// TIA Portal project "Abschulss_Projekt" (V18)
// Vorlageprojekt für das Buch mit Zielsystem S7-1200

(* hardware
DEVICE "S7-1500/ET200MP-Station_1"  S7-1500 station
   slot 0: "Profilschiene_0"  Rack  6ES7 590-1***0-0AA0
   slot 1: "PLC_1"  CPU 1511-1 PN  6ES7 511-1AK00-0AB0  V1.8
      slot 3: "CPU-Display_1"  6ES7591-1AA00-0AA0
      slot 32768: "PROFINET-Schnittstelle_1"  X1
         slot 32769: "Port_1"  X1 P1
         slot 32770: "Port_2"  X1 P2
DEVICE "HMI_1"  KTP900 Basic PN
   slot 0: "HMI_1"  KTP900 Basic PN  6AV2 123-2JB03-0AX0  17.0.0.0
   slot 1: "HMI_RT_1"  KTP900 Basic PN  6AV2 123-2JB03-0AX0  17.0.0.0
   slot 5: "HMI_1.IE_CP_1"  PROFINET Interface  17.0.0.0
      slot 1: "PROFINET Schnittstelle_1"  PROFINET Interface
         slot 1: "Port_1"  Port
*)

// ===== PLC "PLC_1"  CPU 1511-1 PN =====

VAR_GLOBAL   // PLC tag table "Aktor"
   "FACTORY I/O (Reset)(1)" AT %Q8.0 : Bool;
   "Band_Base_1" AT %Q0.0 : Bool;
   "Band_Base_2" AT %Q0.1 : Bool;
   "Band_Base_4" AT %Q0.2 : Bool;
   "Band_Base_6_Gripper" AT %Q0.3 : Bool;
   "R1_Warning_Light" AT %Q0.4 : Bool;
   "R2_Warning_Light" AT %Q0.5 : Bool;
   "Band_Lid_1" AT %Q1.0 : Bool;
   "Band_Lid_2" AT %Q1.1 : Bool;
   "Band_Lid_4" AT %Q1.2 : Bool;
   "Band_Lid_6_Gripper" AT %Q1.3 : Bool;
   "Band_Palletizer_1" AT %Q1.4 : Bool;
   "Loading_to_Crane_Conveyor" AT %Q1.5 : Bool;
   "Emitter_Euro_Palette" AT %Q1.6 : Bool;
   "Curved_Band_Base_3" AT %Q1.7 : Bool;
   "Curved_Band_Base_5" AT %Q2.0 : Bool;
   "Curved_Band_Lid_3" AT %Q2.1 : Bool;
   "Curved_Band_Lid_5" AT %Q2.2 : Bool;
   "Emitter_Base" AT %Q2.3 : Bool;
   "Emitter_Lid" AT %Q2.4 : Bool;
   "Emitter_Package_M" AT %Q2.5 : Bool;
   "Grip_Gripper" AT %Q2.6 : Bool;
   "Palletizer_1_Push" AT %Q2.7 : Bool;
   "Palletizer_1_Turn" AT %Q3.0 : Bool;
   "Palletizer_1_Clamp" AT %Q3.1 : Bool;
   "Palletizer_1_Belt_Plus" AT %Q3.2 : Bool;
   "Palletizer_1_Chain_Plus" AT %Q3.3 : Bool;
   "Palletizer_1_Open_Plate" AT %Q3.4 : Bool;
   "Palletizer_1_Belt_Minuns" AT %Q3.5 : Bool;
   "Palletizer_1_Chain_Minus" AT %Q3.6 : Bool;
   "Palletizer_1_Elevator_Plus" AT %Q3.7 : Bool;
   "Palletizer_1_Elevator_Minus" AT %Q4.0 : Bool;
   "Palletizer_1_Elevator_Move_to_Limit" AT %Q4.1 : Bool;
   "Press_Base" AT %Q4.2 : Bool;
   "Press_Base_Positioner_0_Raise" AT %Q4.3 : Bool;
   "Press_Lid" AT %Q4.4 : Bool;
   "Press_Lid_Positioner_0_Raise" AT %Q4.5 : Bool;
   "R1_Stop" AT %Q4.6 : Bool;
   "R2_Stop" AT %Q4.7 : Bool;
   "R1_Reset" AT %Q5.0 : Bool;
   "R1_Start" AT %Q5.1 : Bool;
   "R2_Reset" AT %Q5.2 : Bool;
   "R2_Start" AT %Q5.3 : Bool;
   "R1_Produce_Lids" AT %Q5.4 : Bool;
   "R2_Produce_Base" AT %Q5.5 : Bool;
   "Remover_Product" AT %Q5.6 : Bool;
   "StackerCrane_1_Left" AT %Q5.7 : Bool;
   "StackerCrane_1_Lift" AT %Q6.0 : Bool;
   "StackerCrane_1_Right" AT %Q6.1 : Bool;
   "X_Move_Gripper" AT %Q6.2 : Bool;
   "Z_Move_Gripper" AT %Q6.3 : Bool;
   "StackerCrane_1_Target_1_Position" AT %QD100 : DInt;
   "Loading_Conveyor_Remover" AT %Q6.4 : Bool;
   "Remove_Euro_Palete" AT %Q6.5 : Bool;
END_VAR

VAR_GLOBAL   // PLC tag table "Merker"
   "Reset" AT %M15.0 : Bool;
END_VAR

VAR_GLOBAL   // PLC tag table "Sensor"
   "FACTORY I/O (Reset)" AT %I4.2 : Bool;
   "LT_Colour_Sorter" AT %I0.0 : Bool;
   "LT_Emitter_Base" AT %I0.1 : Bool;
   "LT_Emitter_Lid" AT %I0.2 : Bool;
   "LT_Palletizer" AT %I0.3 : Bool;
   "LT_Press_Base_Gripper" AT %I0.4 : Bool;
   "LT_Press_Lid_Gripper" AT %I0.5 : Bool;
   "Palletizer_1_Clamped" AT %I0.6 : Bool;
   "Palletizer_1_Plate_Limit" AT %I0.7 : Bool;
   "Palletizer_1_Pusher_Limit" AT %I1.0 : Bool;
   "Palletizer_1_Elevator_Moving" AT %I1.1 : Bool;
   "Palletizer_1_Elevator_Back_Limit" AT %I1.2 : Bool;
   "Palletizer_1_Elevator_Front_Limit" AT %I1.3 : Bool;
   "Press_Base_Positioner_0_Limit" AT %I1.4 : Bool;
   "Press_Lid_Positioner_0_Limit" AT %I1.5 : Bool;
   "R1_Opened" AT %I1.6 : Bool;
   "R2_Opened" AT %I1.7 : Bool;
   "R1_Is_Busy" AT %I2.0 : Bool;
   "R2_Is_Busy" AT %I2.1 : Bool;
   "R1_Has_Error" AT %I2.2 : Bool;
   "R2_Has_Error" AT %I2.3 : Bool;
   "Sensor_Base_fixiert" AT %I2.4 : Bool;
   "Sensor_Greifer_Teilerkennung" AT %I2.5 : Bool;
   "Sensor_Lid_fixiert" AT %I2.6 : Bool;
   "StackerCrane_1_Moving_X" AT %I2.7 : Bool;
   "StackerCrane_1_Moving_Z" AT %I3.0 : Bool;
   "StackerCrane_1_Left_Limit" AT %I3.1 : Bool;
   "StackerCrane_1_Right_Limit" AT %I3.2 : Bool;
   "X_Move_Sensor" AT %I3.3 : Bool;
   "Z_Move_Sensor" AT %I3.4 : Bool;
   "LT_Crane_Feed" AT %I3.5 : Bool;
   "StackerCrane_1_Middle_Limit" AT %I3.6 : Bool;
   "R1_Progress" AT %ID100 : DInt;
   "R2_Progress" AT %ID104 : DInt;
   "Vision_Sensor_Base" AT %ID108 : DInt;
   "Vision_Sensor_Lid" AT %ID112 : DInt;
   "LT_Remove_Palete" AT %I3.7 : Bool;
END_VAR

// folder: 01_Common

DATA_BLOCK "FB_Reset PLC und FactoryIO_DB"   // DB1
{ S7_Optimized_Access := 'TRUE' }
VERSION : 0.1
// stored: InstanceOfName FB_Reset PLC und FactoryIO
"FB_Reset PLC und FactoryIO"
BEGIN
END_DATA_BLOCK

DATA_BLOCK "DB_Global"   // DB2
{ S7_Optimized_Access := 'TRUE' }
VERSION : 0.1
   VAR
      Plant_Enabled : Bool := false;
      Warehouse_Full : Bool;
      Production_Enable : Bool;
      HMI_LidStatus : USInt;
      HMI_BaseStatus : USInt;
      HMI_WarehouseStatus : USInt;
      HMI_Status_OK : Bool;
      HMI_OccupiedPositions : DInt;
      HMI_FreePositions : DInt;
      HMI_TotalPackages : DInt;
      HMI_AlarmWord : Word;
      HMI_AckWord : Word;
   END_VAR
BEGIN
END_DATA_BLOCK

DATA_BLOCK "FB_ProductTracking_DB"   // DB3
{ S7_Optimized_Access := 'TRUE' }
VERSION : 0.1
// stored: InstanceOfName FB_ProductTracking
"FB_ProductTracking"
BEGIN
END_DATA_BLOCK

// folder: 02_Production

DATA_BLOCK "FB_LidCenter_DB"   // DB9
{ S7_Optimized_Access := 'TRUE' }
VERSION : 0.1
// stored: InstanceOfName FB_LidProduction
"FB_LidProduction"
BEGIN
END_DATA_BLOCK

DATA_BLOCK "FB_BaseCenter_DB"   // DB10
{ S7_Optimized_Access := 'TRUE' }
VERSION : 0.1
// stored: InstanceOfName FB_BaseProduction
"FB_BaseProduction"
BEGIN
END_DATA_BLOCK

// folder: 03_Assembly

DATA_BLOCK "FB_Assembly_DB"   // DB11
{ S7_Optimized_Access := 'TRUE' }
VERSION : 0.1
// stored: InstanceOfName FB_Assembly
"FB_Assembly"
BEGIN
END_DATA_BLOCK

DATA_BLOCK "FB_AssemblyActors_DB"   // DB12
{ S7_Optimized_Access := 'TRUE' }
VERSION : 0.1
// stored: InstanceOfName FB_AssemblyActors
"FB_AssemblyActors"
BEGIN
END_DATA_BLOCK

// folder: 04_Palletizer

DATA_BLOCK "FB_Palletizer_DB"   // DB13
{ S7_Optimized_Access := 'TRUE' }
VERSION : 0.1
// stored: InstanceOfName FB_Palletizer
"FB_Palletizer"
BEGIN
END_DATA_BLOCK

// folder: 06_Warehouse

DATA_BLOCK "FB_Warehouse_DB"   // DB14
{ S7_Optimized_Access := 'TRUE' }
VERSION : 0.1
// stored: InstanceOfName FB_Warehouse
"FB_Warehouse"
BEGIN
END_DATA_BLOCK

// folder: 07_HMI

DATA_BLOCK "DB_HMI"   // DB8
{ S7_Optimized_Access := 'TRUE' }
VERSION : 0.1
BEGIN
END_DATA_BLOCK

// folder: 00_Main

ORGANIZATION_BLOCK "Main"   // OB1, FBD, ProgramCycle
TITLE = "Main Program Sweep (Cycle)"
{ S7_Optimized_Access := 'TRUE' }
VERSION : 0.1
   VAR_INPUT
      Initial_Call : Bool;   // Initial call of this OB
      Remanence : Bool;   // =True, if remanent data are available
   END_VAR
BEGIN

REGION Network 1: Factory IO
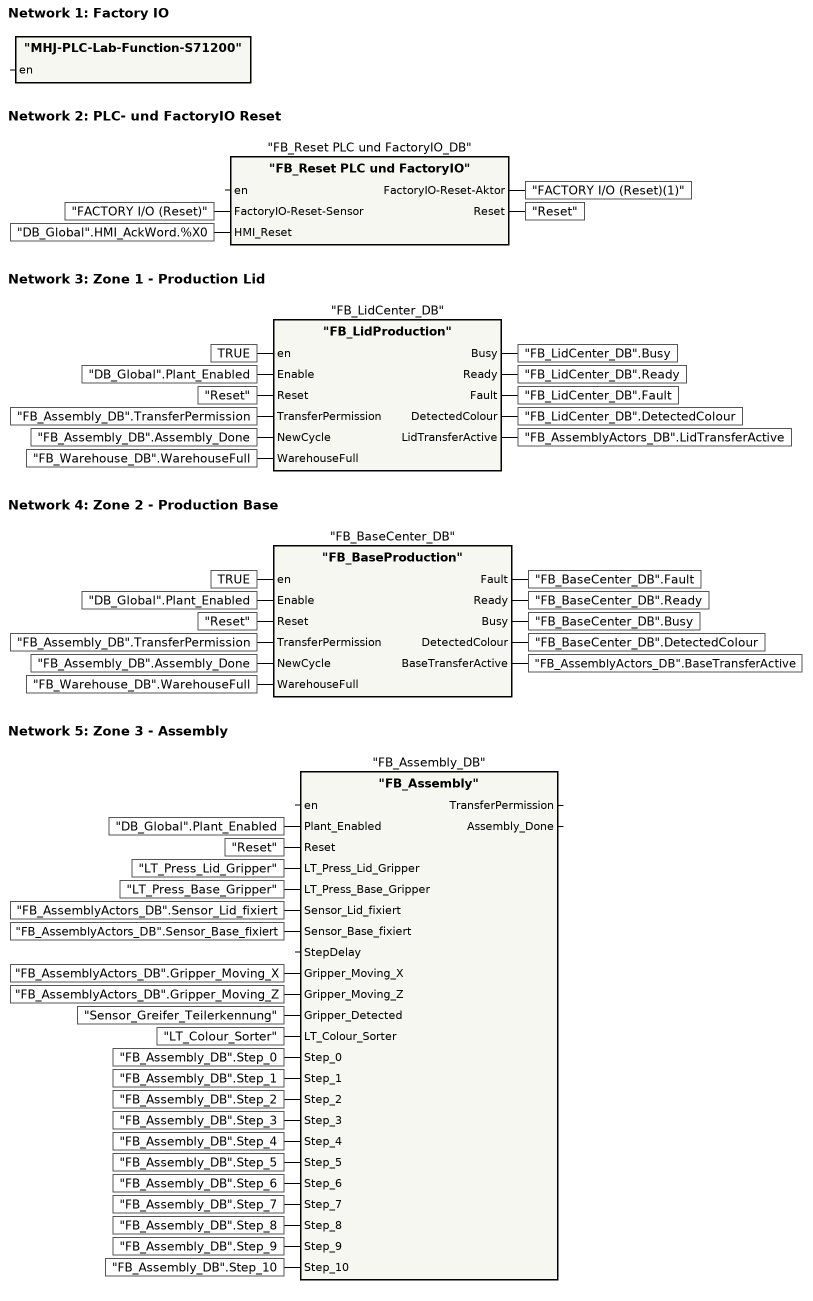
   "MHJ-PLC-Lab-Function-S71200"();
END_REGION

REGION Network 2: PLC- und FactoryIO Reset
   "FB_Reset PLC und FactoryIO_DB"("FactoryIO-Reset-Sensor" := "FACTORY I/O (Reset)",   // "FB_Reset PLC und FactoryIO"
                           HMI_Reset := "DB_Global".HMI_AckWord.%X0,
                           "FactoryIO-Reset-Aktor" => "FACTORY I/O (Reset)(1)",
                           Reset => "Reset");
END_REGION

REGION Network 3: Zone 1 - Production Lid
   IF TRUE THEN
       "FB_LidCenter_DB"(Enable := "DB_Global".Plant_Enabled,   // "FB_LidProduction"
                         Reset := "Reset",
                         TransferPermission := "FB_Assembly_DB".TransferPermission,
                         NewCycle := "FB_Assembly_DB".Assembly_Done,
                         WarehouseFull := "FB_Warehouse_DB".WarehouseFull,
                         Busy => "FB_LidCenter_DB".Busy,
                         Ready => "FB_LidCenter_DB".Ready,
                         Fault => "FB_LidCenter_DB".Fault,
                         DetectedColour => "FB_LidCenter_DB".DetectedColour,
                         LidTransferActive => "FB_AssemblyActors_DB".LidTransferActive);
   END_IF;
END_REGION

REGION Network 4: Zone 2 - Production Base
   IF TRUE THEN
       "FB_BaseCenter_DB"(Enable := "DB_Global".Plant_Enabled,   // "FB_BaseProduction"
                          Reset := "Reset",
                          TransferPermission := "FB_Assembly_DB".TransferPermission,
                          NewCycle := "FB_Assembly_DB".Assembly_Done,
                          WarehouseFull := "FB_Warehouse_DB".WarehouseFull,
                          Fault => "FB_BaseCenter_DB".Fault,
                          Ready => "FB_BaseCenter_DB".Ready,
                          Busy => "FB_BaseCenter_DB".Busy,
                          DetectedColour => "FB_BaseCenter_DB".DetectedColour,
                          BaseTransferActive => "FB_AssemblyActors_DB".BaseTransferActive);
   END_IF;
END_REGION

REGION Network 5: Zone 3 - Assembly
   "FB_Assembly_DB"(Plant_Enabled := "DB_Global".Plant_Enabled,   // "FB_Assembly"
                    Reset := "Reset",
                    LT_Press_Lid_Gripper := "LT_Press_Lid_Gripper",
                    LT_Press_Base_Gripper := "LT_Press_Base_Gripper",
                    Sensor_Lid_fixiert := "FB_AssemblyActors_DB".Sensor_Lid_fixiert,
                    Sensor_Base_fixiert := "FB_AssemblyActors_DB".Sensor_Base_fixiert,
                    Gripper_Moving_X := "FB_AssemblyActors_DB".Gripper_Moving_X,
                    Gripper_Moving_Z := "FB_AssemblyActors_DB".Gripper_Moving_Z,
                    Gripper_Detected := "Sensor_Greifer_Teilerkennung",
                    LT_Colour_Sorter := "LT_Colour_Sorter",
                    Step_0 := "FB_Assembly_DB".Step_0,
                    Step_1 := "FB_Assembly_DB".Step_1,
                    Step_2 := "FB_Assembly_DB".Step_2,
                    Step_3 := "FB_Assembly_DB".Step_3,
                    Step_4 := "FB_Assembly_DB".Step_4,
                    Step_5 := "FB_Assembly_DB".Step_5,
                    Step_6 := "FB_Assembly_DB".Step_6,
                    Step_7 := "FB_Assembly_DB".Step_7,
                    Step_8 := "FB_Assembly_DB".Step_8,
                    Step_9 := "FB_Assembly_DB".Step_9,
                    Step_10 := "FB_Assembly_DB".Step_10);
END_REGION

REGION Network 6: Zone 3 - AssemblyActors
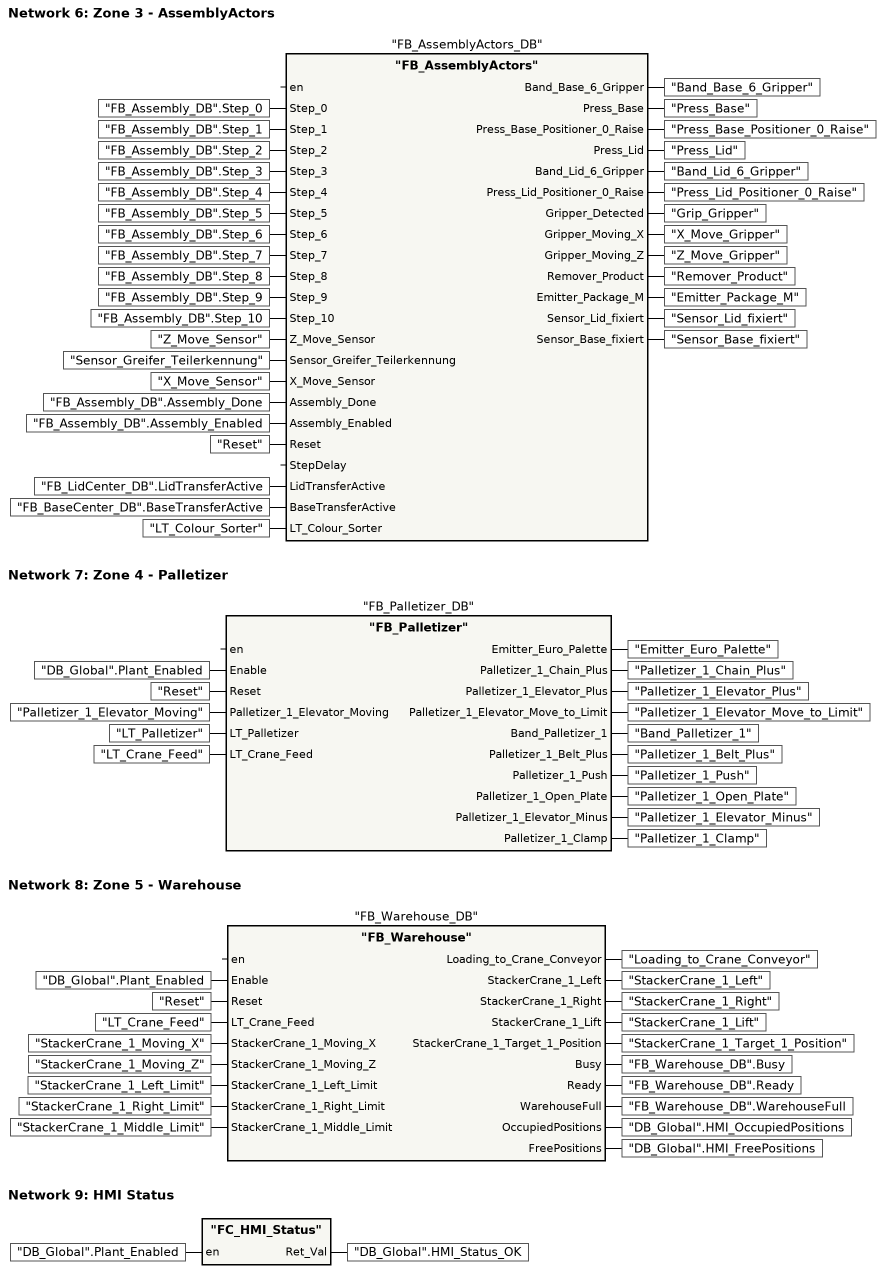
   "FB_AssemblyActors_DB"(Step_0 := "FB_Assembly_DB".Step_0,   // "FB_AssemblyActors"
                          Step_1 := "FB_Assembly_DB".Step_1,
                          Step_2 := "FB_Assembly_DB".Step_2,
                          Step_3 := "FB_Assembly_DB".Step_3,
                          Step_4 := "FB_Assembly_DB".Step_4,
                          Step_5 := "FB_Assembly_DB".Step_5,
                          Step_6 := "FB_Assembly_DB".Step_6,
                          Step_7 := "FB_Assembly_DB".Step_7,
                          Step_8 := "FB_Assembly_DB".Step_8,
                          Step_9 := "FB_Assembly_DB".Step_9,
                          Step_10 := "FB_Assembly_DB".Step_10,
                          Z_Move_Sensor := "Z_Move_Sensor",
                          Sensor_Greifer_Teilerkennung := "Sensor_Greifer_Teilerkennung",
                          X_Move_Sensor := "X_Move_Sensor",
                          Assembly_Done := "FB_Assembly_DB".Assembly_Done,
                          Assembly_Enabled := "FB_Assembly_DB".Assembly_Enabled,
                          Reset := "Reset",
                          LidTransferActive := "FB_LidCenter_DB".LidTransferActive,
                          BaseTransferActive := "FB_BaseCenter_DB".BaseTransferActive,
                          LT_Colour_Sorter := "LT_Colour_Sorter",
                          Band_Base_6_Gripper => "Band_Base_6_Gripper",
                          Press_Base => "Press_Base",
                          Press_Base_Positioner_0_Raise => "Press_Base_Positioner_0_Raise",
                          Press_Lid => "Press_Lid",
                          Band_Lid_6_Gripper => "Band_Lid_6_Gripper",
                          Press_Lid_Positioner_0_Raise => "Press_Lid_Positioner_0_Raise",
                          Gripper_Detected => "Grip_Gripper",
                          Gripper_Moving_X => "X_Move_Gripper",
                          Gripper_Moving_Z => "Z_Move_Gripper",
                          Remover_Product => "Remover_Product",
                          Emitter_Package_M => "Emitter_Package_M",
                          Sensor_Lid_fixiert => "Sensor_Lid_fixiert",
                          Sensor_Base_fixiert => "Sensor_Base_fixiert");
END_REGION

REGION Network 7: Zone 4 - Palletizer
   "FB_Palletizer_DB"(Enable := "DB_Global".Plant_Enabled,   // "FB_Palletizer"
                      Reset := "Reset",
                      Palletizer_1_Elevator_Moving := "Palletizer_1_Elevator_Moving",
                      LT_Palletizer := "LT_Palletizer",
                      LT_Crane_Feed := "LT_Crane_Feed",
                      Emitter_Euro_Palette => "Emitter_Euro_Palette",
                      Palletizer_1_Chain_Plus => "Palletizer_1_Chain_Plus",
                      Palletizer_1_Elevator_Plus => "Palletizer_1_Elevator_Plus",
                      Palletizer_1_Elevator_Move_to_Limit => "Palletizer_1_Elevator_Move_to_Limit",
                      Band_Palletizer_1 => "Band_Palletizer_1",
                      Palletizer_1_Belt_Plus => "Palletizer_1_Belt_Plus",
                      Palletizer_1_Push => "Palletizer_1_Push",
                      Palletizer_1_Open_Plate => "Palletizer_1_Open_Plate",
                      Palletizer_1_Elevator_Minus => "Palletizer_1_Elevator_Minus",
                      Palletizer_1_Clamp => "Palletizer_1_Clamp");
END_REGION

REGION Network 8: Zone 5 - Warehouse
   "FB_Warehouse_DB"(Enable := "DB_Global".Plant_Enabled,   // "FB_Warehouse"
                     Reset := "Reset",
                     LT_Crane_Feed := "LT_Crane_Feed",
                     StackerCrane_1_Moving_X := "StackerCrane_1_Moving_X",
                     StackerCrane_1_Moving_Z := "StackerCrane_1_Moving_Z",
                     StackerCrane_1_Left_Limit := "StackerCrane_1_Left_Limit",
                     StackerCrane_1_Right_Limit := "StackerCrane_1_Right_Limit",
                     StackerCrane_1_Middle_Limit := "StackerCrane_1_Middle_Limit",
                     Loading_to_Crane_Conveyor => "Loading_to_Crane_Conveyor",
                     StackerCrane_1_Left => "StackerCrane_1_Left",
                     StackerCrane_1_Right => "StackerCrane_1_Right",
                     StackerCrane_1_Lift => "StackerCrane_1_Lift",
                     StackerCrane_1_Target_1_Position => "StackerCrane_1_Target_1_Position",
                     Busy => "FB_Warehouse_DB".Busy,
                     Ready => "FB_Warehouse_DB".Ready,
                     WarehouseFull => "FB_Warehouse_DB".WarehouseFull,
                     OccupiedPositions => "DB_Global".HMI_OccupiedPositions,
                     FreePositions => "DB_Global".HMI_FreePositions);
END_REGION

REGION Network 9: HMI Status
   IF "DB_Global".Plant_Enabled THEN "DB_Global".HMI_Status_OK := "FC_HMI_Status"(); END_IF;
END_REGION

REGION Network 10: Product Tracking
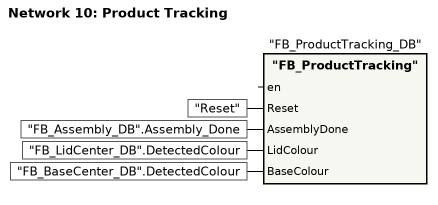
   "FB_ProductTracking_DB"(Reset := "Reset",   // "FB_ProductTracking"
                           AssemblyDone := "FB_Assembly_DB".Assembly_Done,
                           LidColour := "FB_LidCenter_DB".DetectedColour,
                           BaseColour := "FB_BaseCenter_DB".DetectedColour);
END_REGION
END_ORGANIZATION_BLOCK

// folder: 01_Common

FUNCTION_BLOCK "FB_Reset PLC und FactoryIO"   // FB1, FBD
{ S7_Optimized_Access := 'TRUE' }
VERSION : 0.1
   VAR_INPUT
      "FactoryIO-Reset-Sensor" : Bool;
      HMI_Reset : Bool;
   END_VAR
   VAR_OUTPUT
      "FactoryIO-Reset-Aktor" : Bool;
      Reset : Bool;
   END_VAR
   VAR
      M_PLC_reset : Bool;
      "M_PLC-On" : Bool;
   END_VAR
BEGIN

REGION Network 1: PLC- und FactoryIO Reset
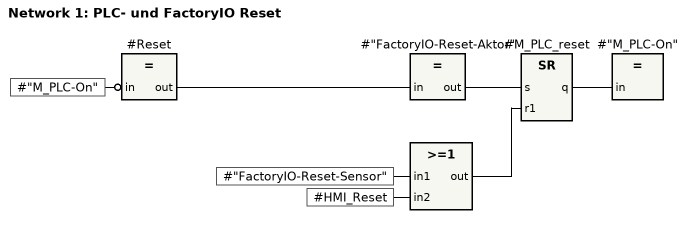
   #Reset := NOT #"M_PLC-On";
   #"FactoryIO-Reset-Aktor" := NOT #"M_PLC-On";
   IF NOT #"M_PLC-On" THEN
       #M_PLC_reset := TRUE;   // SR flip-flop
   END_IF;
   IF #"FactoryIO-Reset-Sensor" OR #HMI_Reset THEN #M_PLC_reset := FALSE; END_IF;
   #"M_PLC-On" := #M_PLC_reset;
END_REGION
END_FUNCTION_BLOCK

FUNCTION_BLOCK "FB_ProductTracking"   // FB8, SCL
{ S7_Optimized_Access := 'TRUE' }
VERSION : 0.1
   VAR_INPUT
      Reset : Bool;
      AssemblyDone : Bool;
      LidColour : Int;
      BaseColour : Int;
   END_VAR
   VAR
      AssemblyDoneOld : Bool;
      Count_BlueBlue : DInt;
      Count_BlueGreen : DInt;
      Count_BlueMetal : DInt;
      Count_GreenBlue : DInt;
      Count_GreenGreen : DInt;
      Count_GreenMetal : DInt;
      Count_MetalBlue : DInt;
      Count_MetalGreen : DInt;
      Count_MetalMetal : DInt;
      CurrentProductType : USInt;
   END_VAR
BEGIN
   // Product Tracking defined BY Base colour + Lid colour:
   IF #Reset THEN
       #CurrentProductType := 0;

       #Count_BlueBlue := 0;
       #Count_BlueGreen := 0;
       #Count_BlueMetal := 0;

       #Count_GreenBlue := 0;
       #Count_GreenGreen := 0;
       #Count_GreenMetal := 0;

       #Count_MetalBlue := 0;
       #Count_MetalGreen := 0;
       #Count_MetalMetal := 0;

       #AssemblyDoneOld := FALSE;
   ELSE

       // Rising edge of AssemblyDone:
       // Count each finished product only once
       IF #AssemblyDone AND NOT #AssemblyDoneOld THEN

           // Accept only valid Vision Sensor colours
           IF (#BaseColour >= 1) AND (#BaseColour <= 3)
               AND (#LidColour >= 1) AND (#LidColour <= 3) THEN

               // Generate product type 1-9
               #CurrentProductType :=
               INT_TO_USINT(((#BaseColour - 1) * 3) + #LidColour);

               // Count product by colour combination.
               CASE #CurrentProductType OF
                   1:
                       #Count_BlueBlue := #Count_BlueBlue + 1;
                   2:
                       #Count_BlueGreen := #Count_BlueGreen + 1;
                   3:
                       #Count_BlueMetal := #Count_BlueMetal + 1;
                   4:
                       #Count_GreenBlue := #Count_GreenBlue + 1;
                   5:
                       #Count_GreenGreen := #Count_GreenGreen + 1;
                   6:
                       #Count_GreenMetal := #Count_GreenMetal + 1;
                   7:
                       #Count_MetalBlue := #Count_MetalBlue + 1;
                   8:
                       #Count_MetalGreen := #Count_MetalGreen + 1;
                   9:
                       #Count_MetalMetal := #Count_MetalMetal + 1;
               END_CASE;
           END_IF;
       END_IF;

       // Store AssemblyDone for rising-edge detection
       #AssemblyDoneOld := #AssemblyDone;
   END_IF;
END_FUNCTION_BLOCK

FUNCTION "FC_VisionDecode" : Void   // FC1, SCL
{ S7_Optimized_Access := 'TRUE' }
VERSION : 0.1
   VAR_INPUT
      VisionValue : DInt;
      IsLid : Bool;
   END_VAR
   VAR_OUTPUT
      Colour : Int;
      Valid : Bool;
   END_VAR
BEGIN
   // Default values
   #Colour := 0;
   #Valid := FALSE;

   // Decode Vision Sensor
   IF #IsLid THEN

       CASE #VisionValue OF
           2:  // Blue Product Lid
               #Colour := 1;
               #Valid := TRUE;

           5:  // Green Product Lid
               #Colour := 2;
               #Valid := TRUE;

           8:  // Metal Product Lid
               #Colour := 3;
               #Valid := TRUE;
       END_CASE;

   ELSE

       CASE #VisionValue OF
           3:  // Blue Product Base
               #Colour := 1;
               #Valid := TRUE;

           6:  // Green Product Base
               #Colour := 2;
               #Valid := TRUE;

           9:  // Metal Product Base
               #Colour := 3;
               #Valid := TRUE;
       END_CASE;

   END_IF;
END_FUNCTION

FUNCTION "MHJ-PLC-Lab-Function-S71200" : Void   // FC9000, SCL
{ S7_Optimized_Access := 'TRUE' }
VERSION : 0.1
   VAR_TEMP
      rdTimeReturn : Int;
      outputTime : DTL;
      SyncVal : Byte;
      forVal : Int;
      forVal_2 : Int;
      Value : Byte;
   END_VAR
   VAR CONSTANT
      CompVal : Byte := 16#34;
      Value_01 : Byte := 16#11;
      Value_01_DW : DWord := 16#A165_D992;
      Value_02_DW : DWord := 16#58BE_4401;
   END_VAR
BEGIN

   #Value:=PEEK(area := 16#82,
        dbNumber := 0,
        byteOffset := 511);
   #Value := #Value + 1;

   POKE(area := 16#82,
        dbNumber := 0,
        byteOffset := 511,
        value := #Value);

   POKE(area:=16#81,
        dbNumber:=0,
        byteOffset:=1016,
        value:=#Value_01_DW);
   POKE(area := 16#81,
        dbNumber := 0,
        byteOffset := 1020,
        value := #Value_02_DW);

   POKE(area := 16#81,
        dbNumber := 0,
        byteOffset := 511,
        value := B#16#00);

   FOR #forVal := 0 TO 120 DO
       FOR #forVal_2:=0 TO 10 DO
           #rdTimeReturn:=RD_SYS_T(#outputTime);
           #rdTimeReturn := WR_SYS_T(#outputTime);
           #rdTimeReturn := RD_SYS_T(#outputTime);
           #rdTimeReturn := WR_SYS_T(#outputTime);
       END_FOR;
       #SyncVal:= PEEK(area := 16#81,
                      dbNumber := 0,
                      byteOffset := 511);
       IF #SyncVal = #CompVal THEN
          GOTO M_1;
       END_IF;
   END_FOR;
   RETURN;

   M_1:
   POKE(area := 16#81,
        dbNumber := 0,
        byteOffset := 511,
        value := B#16#0);
END_FUNCTION

// folder: 02_Production

FUNCTION_BLOCK "FB_BaseProduction"   // FB2, SCL
{ S7_Optimized_Access := 'TRUE' }
VERSION : 0.1
   VAR_INPUT
      Enable : Bool;
      Reset : Bool;
      TransferPermission : Bool;
      NewCycle : Bool;
      WarehouseFull : Bool;
   END_VAR
   VAR_OUTPUT
      Fault : Bool;
      Ready : Bool;
      Busy : Bool;
      DetectedColour : Int;
      BaseTransferActive : Bool;
   END_VAR
   VAR
      State : Int;
      PartColour : Int;
      MachiningStarted : Bool;
      VisionValid : Bool;
   END_VAR
   VAR_TEMP
      DecodedColour : Int;
      DecodedValid : Bool;
   END_VAR
BEGIN
   // Default outputs
   "Emitter_Base" := FALSE;
   "Band_Base_1" := FALSE;
   "Band_Base_2" := FALSE;
   "R2_Start" := FALSE;
   "Curved_Band_Base_3" := FALSE;
   "Band_Base_4" := FALSE;
   "Curved_Band_Base_5" := FALSE;
   #BaseTransferActive := FALSE;
   #DetectedColour := #PartColour;

   // Vision
   "FC_VisionDecode"(
                     VisionValue := "Vision_Sensor_Base",
                     IsLid := FALSE,
                     Colour => #DecodedColour,
                     Valid => #DecodedValid
   );

   // Reset
   IF #Reset THEN
       #State := 0;
       #PartColour := 0;
       #MachiningStarted := FALSE;
   ELSE

       CASE #State OF
               // 0 - Idle
           0:
               #PartColour := 0;
               #MachiningStarted := FALSE;

               IF #Enable
                   AND NOT #WarehouseFull
                   AND NOT "R2_Has_Error" THEN
                   "Emitter_Base" := TRUE;
                   #State := 1;
               END_IF;

               // 1 - Machining
           1:
               "R2_Start" := TRUE;
               "Band_Base_1" := TRUE;
               IF "R2_Is_Busy" THEN
                   #MachiningStarted := TRUE;
               END_IF;
               IF #MachiningStarted
                   AND NOT "R2_Is_Busy" THEN
                   #State := 2;
               END_IF;

               // 2 - Vision
           2:
               "R2_Start" := TRUE;
               "Band_Base_2" := TRUE;
               IF #DecodedValid THEN
                   #PartColour := #DecodedColour;
                   #State := 3;
               END_IF;

               // 3 - Wait for Assembly
           3:
               IF #TransferPermission THEN
                   #State := 4;
               END_IF;

               // 4 - Transfer to Assembly
           4:
               #BaseTransferActive := TRUE;
               "Band_Base_2" := TRUE;
               "Curved_Band_Base_3" := TRUE;
               "Band_Base_4" := TRUE;
               "Curved_Band_Base_5" := TRUE;
               IF #NewCycle THEN
                   #State := 0;
               END_IF;
           ELSE
               #State := 0;
       END_CASE;
   END_IF;
END_FUNCTION_BLOCK

FUNCTION_BLOCK "FB_LidProduction"   // FB3, SCL
{ S7_Optimized_Access := 'TRUE' }
VERSION : 0.1
   VAR_INPUT
      Enable : Bool;
      Reset : Bool;
      TransferPermission : Bool;
      NewCycle : Bool;
      WarehouseFull : Bool;
   END_VAR
   VAR_OUTPUT
      Busy : Bool;
      Ready : Bool;
      Fault : Bool;
      DetectedColour : Int;
      LidTransferActive : Bool;
   END_VAR
   VAR
      State : Int;
      PartColour : Int;
      MachiningStarted : Bool;
      JamFault : Bool;
      TimerVisionJam : TON_TIME;
      TransferState : Int;
   END_VAR
   VAR_TEMP
      DecodedColour : Int;
      DecodedValid : Bool;
   END_VAR
BEGIN
   "R1_Produce_Lids" := TRUE;
   // Default outputs
   "Emitter_Lid" := FALSE;
   "Band_Lid_1" := FALSE;
   "Band_Lid_2" := FALSE;
   "R1_Start" := FALSE;
   "Curved_Band_Lid_3" := FALSE;
   "Band_Lid_4" := FALSE;
   "Curved_Band_Lid_5" := FALSE;
   #LidTransferActive := FALSE;
   #DetectedColour := #PartColour;

   // Vision
   "FC_VisionDecode"(
                     VisionValue := "Vision_Sensor_Lid",
                     IsLid := TRUE,
                     Colour => #DecodedColour,
                     Valid => #DecodedValid
   );

   // Reset
   IF #Reset THEN
       #State := 0;
       #PartColour := 0;
       #MachiningStarted := FALSE;
   ELSE

       CASE #State OF
               // 0 - Idle
           0:
               #PartColour := 0;
               #MachiningStarted := FALSE;
               IF #Enable
                   AND NOT #WarehouseFull
                   AND NOT "R1_Has_Error" THEN
                   "Emitter_Lid" := TRUE;
                   #State := 1;
               END_IF;

               // 1 - Machining
           1:
               "R1_Start" := TRUE;
               "Band_Lid_1" := TRUE;
               IF "R1_Is_Busy" THEN
                   #MachiningStarted := TRUE;
               END_IF;
               IF #MachiningStarted
                   AND NOT "R1_Is_Busy" THEN
                   #State := 2;
               END_IF;

               // 2 - Vision
           2:
               "R1_Start" := TRUE;
               "Band_Lid_2" := TRUE;
               IF #DecodedValid THEN
                   #PartColour := #DecodedColour;
                   #State := 3;
               END_IF;

               // 3 - Wait for Assembly
           3:
               IF #TransferPermission THEN
                   #State := 4;
               END_IF;

               // 4 - Transfer to Assembly
           4:
               #LidTransferActive := TRUE;
               "Band_Lid_2" := TRUE;
               "Curved_Band_Lid_3" := TRUE;
               "Band_Lid_4" := TRUE;
               "Curved_Band_Lid_5" := TRUE;
               IF #NewCycle THEN
                   #State := 0;
               END_IF;
           ELSE
               #State := 0;
       END_CASE;
   END_IF;
END_FUNCTION_BLOCK

// folder: 03_Assembly

FUNCTION_BLOCK "FB_Assembly"   // FB4, FBD
{ S7_Optimized_Access := 'TRUE' }
VERSION : 0.1
   VAR_INPUT
      Plant_Enabled : Bool;
      Reset : Bool;
      LT_Press_Lid_Gripper : Bool;
      LT_Press_Base_Gripper : Bool;
      Sensor_Lid_fixiert : Bool;
      Sensor_Base_fixiert : Bool;
      StepDelay : Time := T#1s;
      Gripper_Moving_X : Bool;
      Gripper_Moving_Z : Bool;
      Gripper_Detected : Bool;
      LT_Colour_Sorter : Bool;
   END_VAR
   VAR_OUTPUT
      TransferPermission : Bool;
      Assembly_Done : Bool;
   END_VAR
   VAR_IN_OUT
      Step_0 : Bool;
      Step_1 : Bool;
      Step_2 : Bool;
      Step_3 : Bool;
      Step_4 : Bool;
      Step_5 : Bool;
      Step_6 : Bool;
      Step_7 : Bool;
      Step_8 : Bool;
      Step_9 : Bool;
      Step_10 : Bool;
   END_VAR
   VAR
      SR_Assembly_Enabled : Bool;
      Assembly_Enabled : Bool;
      TON_Step_1 : TON_TIME;
      TON_Step_2 : TON_TIME;
      TON_Step_3 : TON_TIME;
      TON_Step_4 : TON_TIME;
      TON_Step_5 : TON_TIME;
      TON_Step_6 : TON_TIME;
      TON_Step_7 : TON_TIME;
      TON_Step_8 : TON_TIME;
      TON_Prozess_Ende : TON_TIME;
      Gripper_Moving : Bool;
      SR_LT_Sorter : Bool;
      SR_Base_Arrived : Bool;
      SR_Lid_Arrived : Bool;
      TON_RemoveDelay : TON_TIME;
      TON_Remover : TON_TIME;
      TON_Step_9 : TON_TIME;
   END_VAR
BEGIN

REGION Network 1: Assembly Enable / Reset
   // The Assembly sequence is enabled when the plant is active.
   // A PLC reset disables the Assembly sequence.
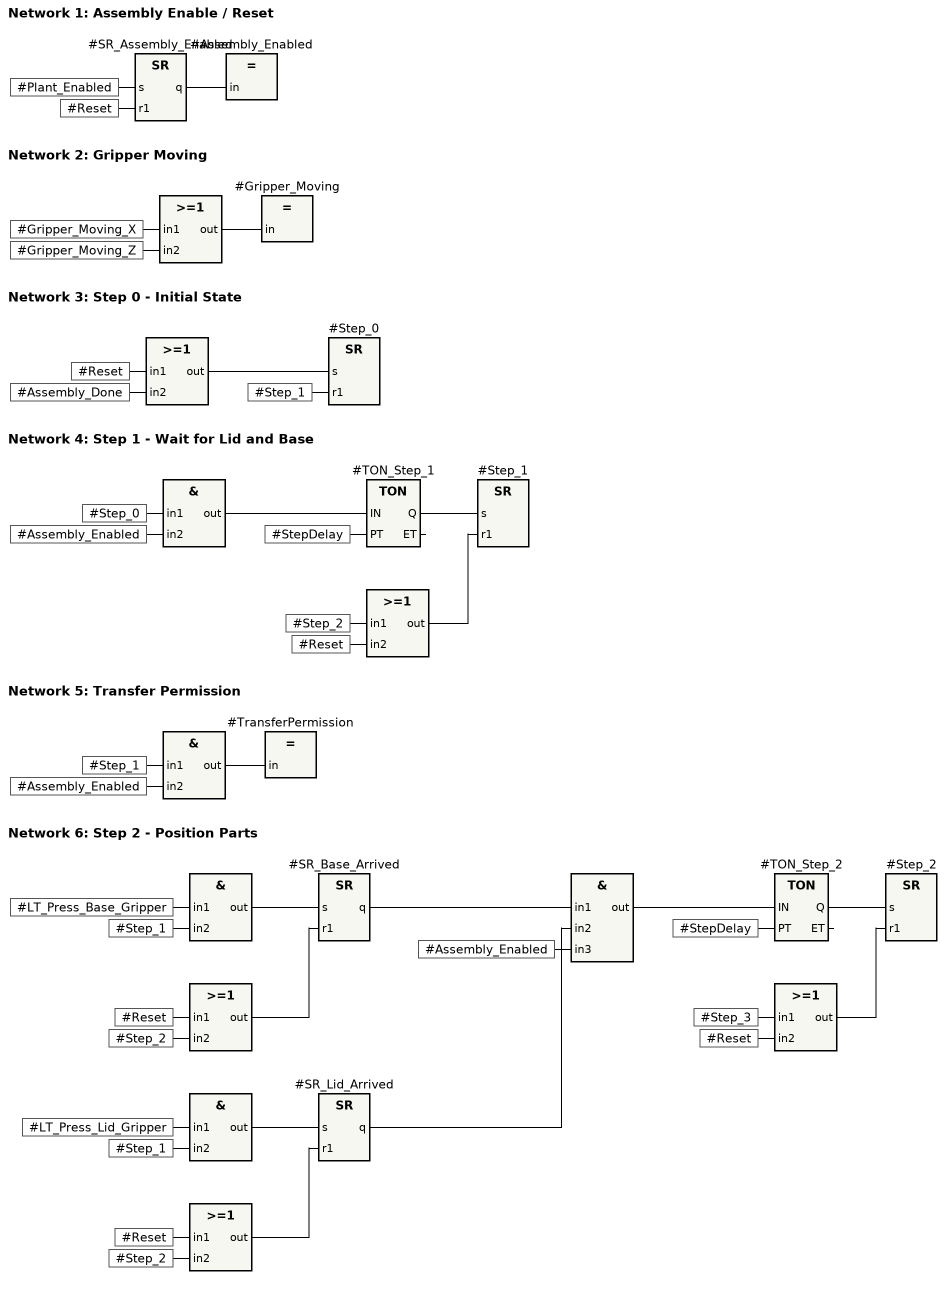
   IF #Plant_Enabled THEN
       #SR_Assembly_Enabled := TRUE;   // SR flip-flop
   END_IF;
   IF #Reset THEN #SR_Assembly_Enabled := FALSE; END_IF;
   #Assembly_Enabled := #SR_Assembly_Enabled;
END_REGION

REGION Network 2: Gripper Moving
   #Gripper_Moving := #Gripper_Moving_X OR #Gripper_Moving_Z;
END_REGION

REGION Network 3: Step 0 - Initial State
   // Initial step of the Assembly sequence.
   // A PLC reset activates Step 0.
   // Step 0 remains active until Step 1 starts.
   IF #Reset OR #Assembly_Done THEN
       #Step_0 := TRUE;   // SR flip-flop
   END_IF;
   IF #Step_1 THEN #Step_0 := FALSE; END_IF;
END_REGION

REGION Network 4: Step 1 - Wait for Lid and Base
   // Step 1 starts when the Assembly sequence is enabled
   // and the initial step is active.
   // The sequence waits for the Lid and Base to arrive.
   #TON_Step_1(IN := #Step_0 AND #Assembly_Enabled, PT := #StepDelay);   // TON
   IF #TON_Step_1.Q THEN
       #Step_1 := TRUE;   // SR flip-flop
   END_IF;
   IF #Step_2 OR #Reset THEN #Step_1 := FALSE; END_IF;
END_REGION

REGION Network 5: Transfer Permission
   // The production modules are allowed to transfer the Lid and Base while the Assembly sequence is waiting for the parts.
   #TransferPermission := #Step_1 AND #Assembly_Enabled;
END_REGION

REGION Network 6: Step 2 - Position Parts
   // Step 2 starts when both Lid and Base have reached the Assembly positioning area.
   // The step remains active until the positioning sequence is completed.
   IF #LT_Press_Base_Gripper AND #Step_1 THEN
       #SR_Base_Arrived := TRUE;   // SR flip-flop
   END_IF;
   IF #Reset OR #Step_2 THEN #SR_Base_Arrived := FALSE; END_IF;
   IF #LT_Press_Lid_Gripper AND #Step_1 THEN
       #SR_Lid_Arrived := TRUE;   // SR flip-flop
   END_IF;
   IF #Reset OR #Step_2 THEN #SR_Lid_Arrived := FALSE; END_IF;
   #TON_Step_2(IN := #SR_Base_Arrived AND #SR_Lid_Arrived AND #Assembly_Enabled, PT := #StepDelay);   // TON
   IF #TON_Step_2.Q THEN
       #Step_2 := TRUE;   // SR flip-flop
   END_IF;
   IF #Step_3 OR #Reset THEN #Step_2 := FALSE; END_IF;
END_REGION

REGION Network 7: Step 3 - Pick Up Lid
   // Step 3 starts when the Lid is correctly positioned and fixed.
   // During this step, the gripper picks up the Lid.
   // The sequence continues when the Lid has been successfully gripped and lifted.
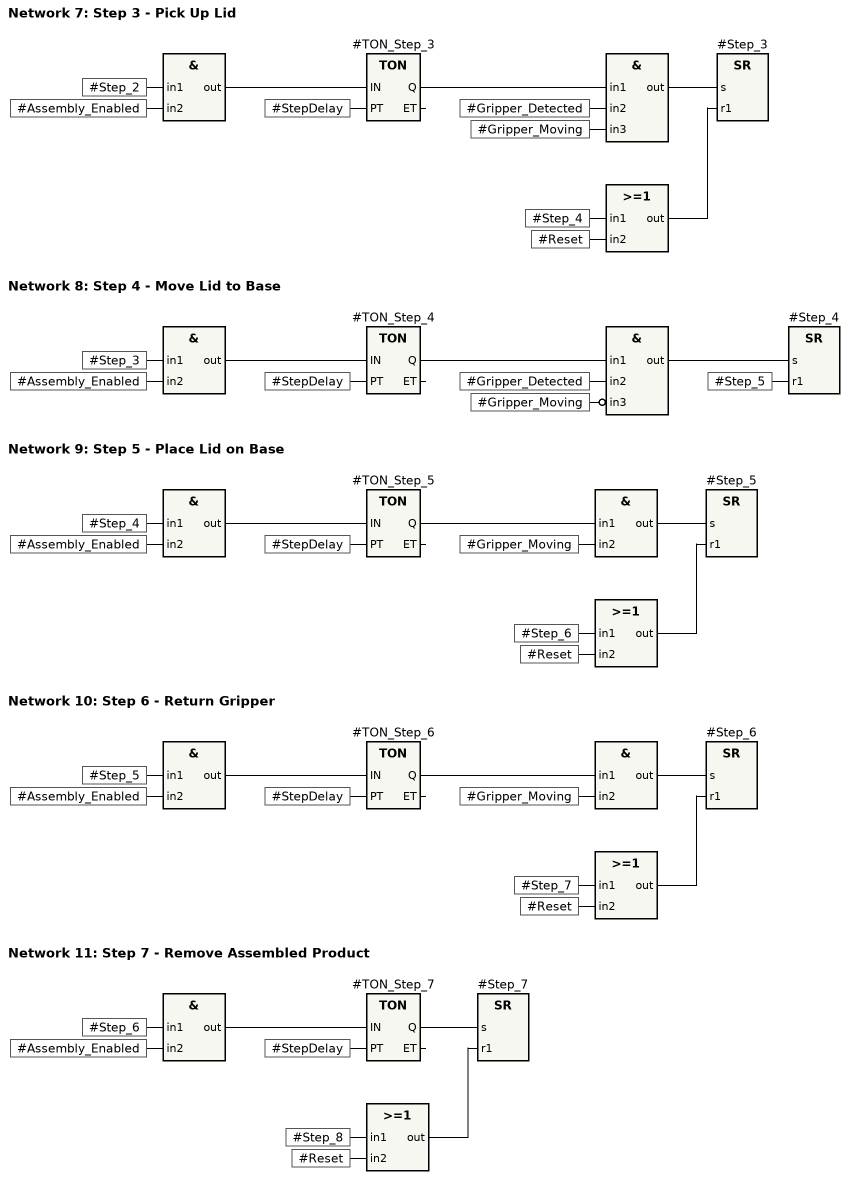
   #TON_Step_3(IN := #Step_2 AND #Assembly_Enabled, PT := #StepDelay);   // TON
   IF #TON_Step_3.Q AND #Gripper_Detected AND #Gripper_Moving THEN
       #Step_3 := TRUE;   // SR flip-flop
   END_IF;
   IF #Step_4 OR #Reset THEN #Step_3 := FALSE; END_IF;
END_REGION

REGION Network 8: Step 4 - Move Lid to Base
   // Step 4 starts after the Lid has been successfully picked up and lifted. During this step, the gripper moves horizontally toward the Base. The sequence continues when the gripper reaches the Base position.
   #TON_Step_4(IN := #Step_3 AND #Assembly_Enabled, PT := #StepDelay);   // TON
   IF #TON_Step_4.Q AND #Gripper_Detected AND NOT #Gripper_Moving THEN
       #Step_4 := TRUE;   // SR flip-flop
   END_IF;
   IF #Step_5 THEN #Step_4 := FALSE; END_IF;
END_REGION

REGION Network 9: Step 5 - Place Lid on Base
   // Step 5 starts when the gripper has reached the position above the Base. During this step, the Lid is lowered onto the Base and released. The sequence continues after the Lid has been successfully placed.
   #TON_Step_5(IN := #Step_4 AND #Assembly_Enabled, PT := #StepDelay);   // TON
   IF #TON_Step_5.Q AND #Gripper_Moving THEN
       #Step_5 := TRUE;   // SR flip-flop
   END_IF;
   IF #Step_6 OR #Reset THEN #Step_5 := FALSE; END_IF;
END_REGION

REGION Network 10: Step 6 - Return Gripper
   // Step 6 starts after the Lid has been successfully placed on the Base and released. During this step, the gripper returns to its home position. The sequence continues when the gripper has reached the home position.
   #TON_Step_6(IN := #Step_5 AND #Assembly_Enabled, PT := #StepDelay);   // TON
   IF #TON_Step_6.Q AND #Gripper_Moving THEN
       #Step_6 := TRUE;   // SR flip-flop
   END_IF;
   IF #Step_7 OR #Reset THEN #Step_6 := FALSE; END_IF;
END_REGION

REGION Network 11: Step 7 - Remove Assembled Product
   // Step 7 starts when the gripper has returned to its home position. During this step, the assembled product is removed and the package is prepared for emission. The sequence continues when the product removal is confirmed.
   #TON_Step_7(IN := #Step_6 AND #Assembly_Enabled, PT := #StepDelay);   // TON
   IF #TON_Step_7.Q THEN
       #Step_7 := TRUE;   // SR flip-flop
   END_IF;
   IF #Step_8 OR #Reset THEN #Step_7 := FALSE; END_IF;
END_REGION

REGION Network 12: Step 8 - Remove asembled Product
   // Step 8 starts after the assembled product has been removed. During this step, one package is emitted for the completed product. The sequence continues when the package emission is confirmed.
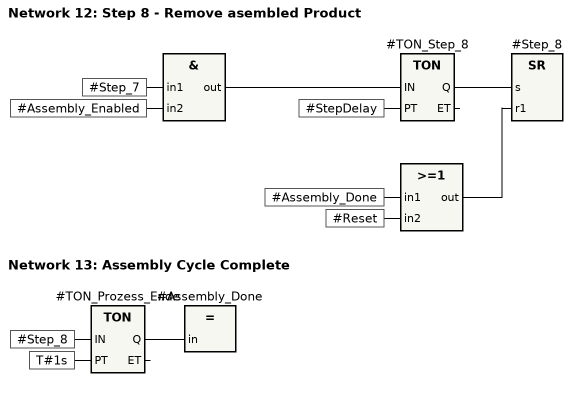
   #TON_Step_8(IN := #Step_7 AND #Assembly_Enabled, PT := #StepDelay);   // TON
   IF #TON_Step_8.Q THEN
       #Step_8 := TRUE;   // SR flip-flop
   END_IF;
   IF #Assembly_Done OR #Reset THEN #Step_8 := FALSE; END_IF;
END_REGION

REGION Network 13: Assembly Cycle Complete
   // The Assembly cycle is completed after Step 8 has successfully emitted the package. The completion signal terminates Step 8 and returns the sequence to the initial state, ready for the next Lid/Base assembly cycle.
   #TON_Prozess_Ende(IN := #Step_8, PT := T#1s);   // TON
   #Assembly_Done := #TON_Prozess_Ende.Q;
END_REGION
END_FUNCTION_BLOCK

FUNCTION_BLOCK "FB_AssemblyActors"   // FB7, FBD
{ S7_Optimized_Access := 'TRUE' }
VERSION : 0.1
   VAR_INPUT
      Step_0 : Bool;
      Step_1 : Bool;
      Step_2 : Bool;
      Step_3 : Bool;
      Step_4 : Bool;
      Step_5 : Bool;
      Step_6 : Bool;
      Step_7 : Bool;
      Step_8 : Bool;
      Step_9 : Bool;
      Step_10 : Bool;
      Z_Move_Sensor : Bool;
      Sensor_Greifer_Teilerkennung : Bool;
      X_Move_Sensor : Bool;
      Assembly_Done : Bool;
      Assembly_Enabled : Bool;
      Reset : Bool;
      StepDelay : Time := T#1s;
      LidTransferActive : Bool;
      BaseTransferActive : Bool;
      LT_Colour_Sorter : Bool;
   END_VAR
   VAR_OUTPUT
      Band_Base_6_Gripper : Bool;
      Press_Base : Bool;
      Press_Base_Positioner_0_Raise : Bool;
      Press_Lid : Bool;
      Band_Lid_6_Gripper : Bool;
      Press_Lid_Positioner_0_Raise : Bool;
      Gripper_Detected : Bool;
      Gripper_Moving_X : Bool;
      Gripper_Moving_Z : Bool;
      Remover_Product : Bool;
      Emitter_Package_M : Bool;
      Sensor_Lid_fixiert : Bool;
      Sensor_Base_fixiert : Bool;
   END_VAR
   VAR
      SR_Band_Lid : Bool;
      SR_Press_Lid : Bool;
      SR_Press_Base : Bool;
      SR_Gripper_Z : Bool;
      SR_Gripper_Grip : Bool;
      TON_Greifer_Vor_Reset : TON_TIME;
      SR_Gripper_X : Bool;
      SR_Band_Base : Bool;
      R_TRIG : R_TRIG;
   END_VAR
   VAR_TEMP   // added for the SCL form of the ladder/FBD networks
      _w1 : Bool;
   END_VAR
BEGIN

REGION Network 1: Band Lid
   // The Lid and Base conveyors transport the produced parts from the production modules to the Assembly station while Step 1 is active.
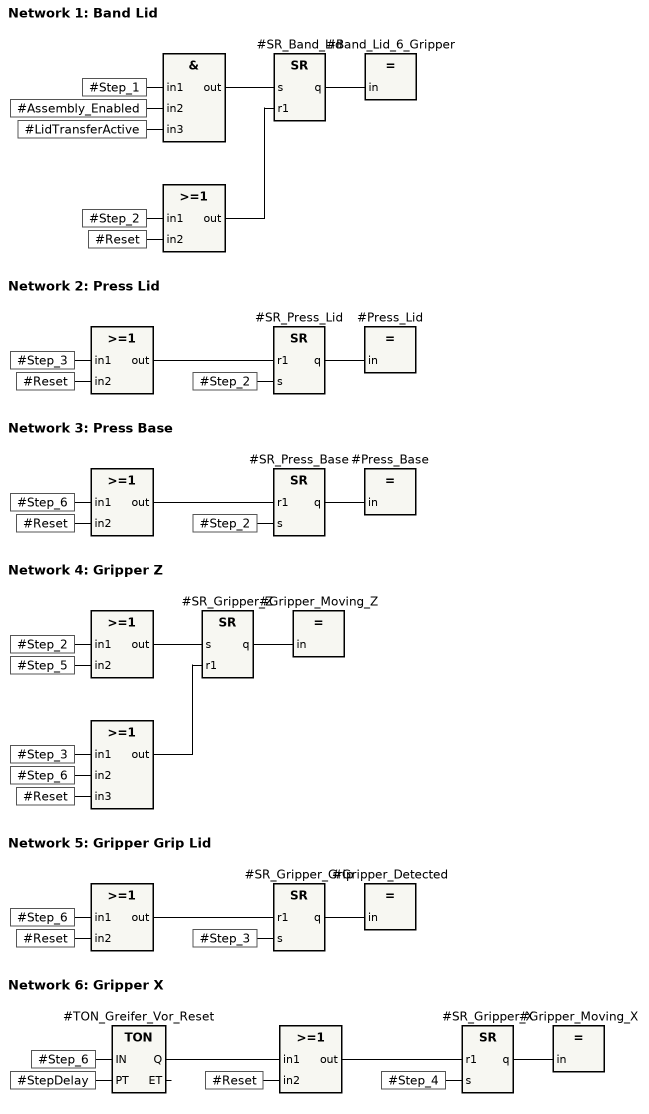
   IF #Step_1 AND #Assembly_Enabled AND #LidTransferActive THEN
       #SR_Band_Lid := TRUE;   // SR flip-flop
   END_IF;
   IF #Step_2 OR #Reset THEN #SR_Band_Lid := FALSE; END_IF;
   #Band_Lid_6_Gripper := #SR_Band_Lid;
END_REGION

REGION Network 2: Press Lid
   IF #Step_2 THEN
       #SR_Press_Lid := TRUE;   // SR flip-flop
   END_IF;
   IF #Step_3 OR #Reset THEN #SR_Press_Lid := FALSE; END_IF;
   #Press_Lid := #SR_Press_Lid;
END_REGION

REGION Network 3: Press Base
   IF #Step_2 THEN
       #SR_Press_Base := TRUE;   // SR flip-flop
   END_IF;
   IF #Step_6 OR #Reset THEN #SR_Press_Base := FALSE; END_IF;
   #Press_Base := #SR_Press_Base;
END_REGION

REGION Network 4: Gripper Z
   IF #Step_2 OR #Step_5 THEN
       #SR_Gripper_Z := TRUE;   // SR flip-flop
   END_IF;
   IF #Step_3 OR #Step_6 OR #Reset THEN #SR_Gripper_Z := FALSE; END_IF;
   #Gripper_Moving_Z := #SR_Gripper_Z;
END_REGION

REGION Network 5: Gripper Grip Lid
   IF #Step_3 THEN
       #SR_Gripper_Grip := TRUE;   // SR flip-flop
   END_IF;
   IF #Step_6 OR #Reset THEN #SR_Gripper_Grip := FALSE; END_IF;
   #Gripper_Detected := #SR_Gripper_Grip;
END_REGION

REGION Network 6: Gripper X
   #TON_Greifer_Vor_Reset(IN := #Step_6, PT := #StepDelay);   // TON
   IF #Step_4 THEN
       #SR_Gripper_X := TRUE;   // SR flip-flop
   END_IF;
   IF #TON_Greifer_Vor_Reset.Q OR #Reset THEN #SR_Gripper_X := FALSE; END_IF;
   #Gripper_Moving_X := #SR_Gripper_X;
END_REGION

REGION Network 7: Band Base
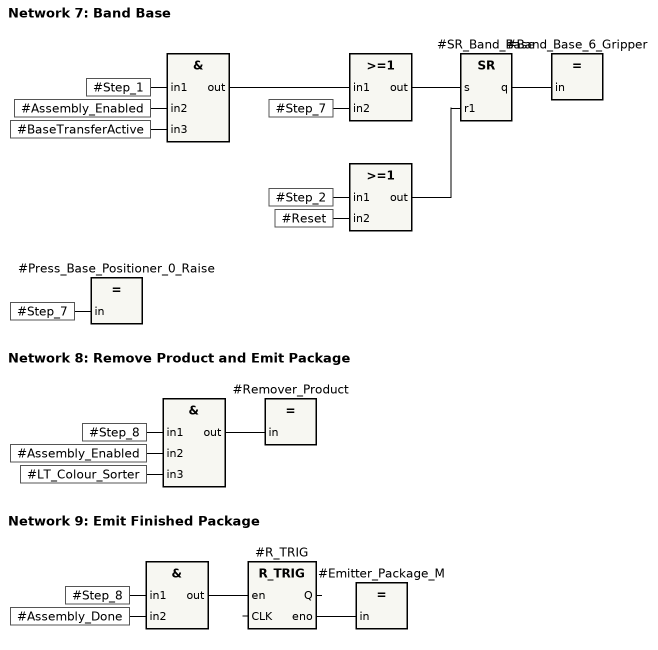
   IF (#Step_1 AND #Assembly_Enabled AND #BaseTransferActive) OR #Step_7 THEN
       #SR_Band_Base := TRUE;   // SR flip-flop
   END_IF;
   IF #Step_2 OR #Reset THEN #SR_Band_Base := FALSE; END_IF;
   #Band_Base_6_Gripper := #SR_Band_Base;
   #Press_Base_Positioner_0_Raise := #Step_7;
END_REGION

REGION Network 8: Remove Product and Emit Package
   #Remover_Product := #Step_8 AND #Assembly_Enabled AND #LT_Colour_Sorter;
END_REGION

REGION Network 9: Emit Finished Package
   // ENO of a box is taken as its EN; it also drops when the box reports an error
   #_w1 := #Step_8 AND #Assembly_Done;
   IF #_w1 THEN
       #R_TRIG();   // R_TRIG
   END_IF;
   #Emitter_Package_M := #_w1;
END_REGION
END_FUNCTION_BLOCK

// folder: 04_Palletizer

FUNCTION_BLOCK "FB_Palletizer"   // FB5, SCL
{ S7_Optimized_Access := 'TRUE' }
VERSION : 0.1
   VAR_INPUT
      Enable : Bool;
      Reset : Bool;
      Palletizer_1_Elevator_Moving : Bool;
      LT_Palletizer : Bool;
      LT_Crane_Feed : Bool;
   END_VAR
   VAR_OUTPUT
      Emitter_Euro_Palette : Bool;
      Palletizer_1_Chain_Plus : Bool;
      Palletizer_1_Elevator_Plus : Bool;
      Palletizer_1_Elevator_Move_to_Limit : Bool;
      Band_Palletizer_1 : Bool;
      Palletizer_1_Belt_Plus : Bool;
      Palletizer_1_Push : Bool;
      Palletizer_1_Open_Plate : Bool;
      Palletizer_1_Elevator_Minus : Bool;
      Palletizer_1_Clamp : Bool;
   END_VAR
   VAR
      State : Int;
      ElevatorStarted : Bool;
      PackageCounter : Int;
      LT_Palletizer_Old : Bool;
      PushCounter : Int;
      TimerPalletSettle : TON_TIME;
      TimerBeforePush : TON_TIME;
      TimerPush : TON_TIME;
      TimerPlateOpen : TON_TIME;
      TimerClamp : TON_TIME;
   END_VAR
   VAR_TEMP
      Busy : Bool;
      Ready : Bool;
   END_VAR
BEGIN
   // Default outputs
   #Emitter_Euro_Palette := FALSE;
   #Band_Palletizer_1 := FALSE;
   #Palletizer_1_Belt_Plus := FALSE;
   #Palletizer_1_Push := FALSE;
   #Palletizer_1_Open_Plate := FALSE;
   #Palletizer_1_Clamp := FALSE;
   #Palletizer_1_Elevator_Plus := FALSE;
   #Palletizer_1_Elevator_Minus := FALSE;
   #Palletizer_1_Elevator_Move_to_Limit := FALSE;
   #Palletizer_1_Chain_Plus := FALSE;

   // Timers
   #TimerPalletSettle(
                      IN := (#State = 0) AND #Enable,
                      PT := T#2s
   );

   #TimerBeforePush(
                    IN := (#State = 20) AND (#PackageCounter >= 2),
                    PT := T#3s
   );

   #TimerPush(
              IN := (#State = 30),
              PT := T#1s
   );

   #TimerPlateOpen(
                   IN := (#State = 40),
                   PT := T#7s
   );


   // Reset
   IF #Reset THEN
       #State := 0;
       #PackageCounter := 0;
       #PushCounter := 0;
       #LT_Palletizer_Old := FALSE;
       #ElevatorStarted := FALSE;
   ELSE

       // Count arriving packages
       IF (#State = 20)
           AND #LT_Palletizer
           AND NOT #LT_Palletizer_Old THEN
           #PackageCounter := #PackageCounter + 1;
       END_IF;


       CASE #State OF

               // 0 - Create empty Euro pallet
           0:
               IF #Enable THEN

                   #PackageCounter := 0;
                   #PushCounter := 0;
                   #ElevatorStarted := FALSE;
                   #Emitter_Euro_Palette := TRUE;

                   IF #TimerPalletSettle.Q THEN
                       #State := 10;
                   END_IF;
               END_IF;

               // 10 - Raise empty pallet
           10:
               #Palletizer_1_Elevator_Plus := TRUE;
               #Palletizer_1_Elevator_Move_to_Limit := TRUE;

               IF #Palletizer_1_Elevator_Moving THEN
                   #ElevatorStarted := TRUE;
               END_IF;

               IF #ElevatorStarted
                   AND NOT #Palletizer_1_Elevator_Moving THEN
                   #ElevatorStarted := FALSE;
                   #PackageCounter := 0;
                   #PushCounter := 0;
                   #State := 20;
               END_IF;

               // 20 - Receive two packages
           20:
               #Band_Palletizer_1 := TRUE;
               #Palletizer_1_Belt_Plus := TRUE;

               IF (#PackageCounter >= 2)
                   AND #TimerBeforePush.Q THEN
                   #State := 30;
               END_IF;

               // 30 - Push package pair
           30:
               #Palletizer_1_Push := TRUE;

               IF #TimerPush.Q THEN
                   #PackageCounter := 0;
                   #PushCounter := #PushCounter + 1;
                   IF #PushCounter >= 2 THEN
                       #State := 40;
                   ELSE
                       #State := 20;
                   END_IF;
               END_IF;

               // 40 - Open plate and release packages
           40:
               #Palletizer_1_Open_Plate := TRUE;
               // Hold packages during the first 2 seconds
               #Palletizer_1_Clamp :=
               (#TimerPlateOpen.ET < T#2s);

               IF #TimerPlateOpen.Q THEN
                   #ElevatorStarted := FALSE;
                   #State := 60;
               END_IF;

               // 60 - Lower completed pallet
           60:
               #Palletizer_1_Open_Plate := TRUE;
               #Palletizer_1_Elevator_Minus := TRUE;
               #Palletizer_1_Elevator_Move_to_Limit := TRUE;

               IF #Palletizer_1_Elevator_Moving THEN
                   #ElevatorStarted := TRUE;
               END_IF;

               IF #ElevatorStarted
                   AND NOT #Palletizer_1_Elevator_Moving THEN
                   #ElevatorStarted := FALSE;
                   #State := 70;
               END_IF;

               // 70 - Transfer pallet to Warehouse
           70:
               #Palletizer_1_Chain_Plus := TRUE;
               IF #LT_Crane_Feed THEN
                   #State := 0;
               END_IF;
           ELSE
               #State := 0;
       END_CASE;
       // Store previous light sensor state
       #LT_Palletizer_Old := #LT_Palletizer;
   END_IF;
END_FUNCTION_BLOCK

// folder: 06_Warehouse

FUNCTION_BLOCK "FB_Warehouse"   // FB6, SCL
{ S7_Optimized_Access := 'TRUE' }
VERSION : 0.1
   VAR_INPUT
      Enable : Bool;
      Reset : Bool;
      LT_Crane_Feed : Bool;
      StackerCrane_1_Moving_X : Bool;
      StackerCrane_1_Moving_Z : Bool;
      StackerCrane_1_Left_Limit : Bool;
      StackerCrane_1_Right_Limit : Bool;
      StackerCrane_1_Middle_Limit : Bool;
   END_VAR
   VAR_OUTPUT
      Loading_to_Crane_Conveyor : Bool;
      StackerCrane_1_Left : Bool;
      StackerCrane_1_Right : Bool;
      StackerCrane_1_Lift : Bool;
      StackerCrane_1_Target_1_Position : DInt;
      Busy : Bool;
      Ready : Bool;
      WarehouseFull : Bool;
      OccupiedPositions : Int;
      FreePositions : Int;
   END_VAR
   VAR
      State : Int;
      NextPosition : DInt;
      MovementStarted : Bool;
      TimerLiftUp : TON_TIME;
      TimerLiftDown : TON_TIME;
      TimerDeposit : TON_TIME;
   END_VAR
BEGIN
   // Warehouse position counters
   IF #State = 7 THEN
       #OccupiedPositions := 54;
       #FreePositions := 0;
   ELSE
       #OccupiedPositions := #NextPosition - 1;
       #FreePositions := 54 - #OccupiedPositions;
   END_IF;
   // Deposit timer
   #TimerDeposit(
                 IN := (#State = 4),
                 PT := T#2s
   );

   // Reset
   IF #Reset THEN
       #State := 0;
       #NextPosition := 1;
       #MovementStarted := FALSE;
       #Loading_to_Crane_Conveyor := FALSE;
       #StackerCrane_1_Left := FALSE;
       #StackerCrane_1_Right := FALSE;
       #StackerCrane_1_Lift := FALSE;
       #StackerCrane_1_Target_1_Position := 0;
   ELSE
       // Status
       #Ready := (#State = 0);
       #Busy := (#State > 0) AND (#State < 7);
       #WarehouseFull := (#State = 7);
       CASE #State OF
               // 0 - Wait for pallet
           0:
               #StackerCrane_1_Target_1_Position := 0;
               IF #Enable THEN
                   #Loading_to_Crane_Conveyor := TRUE;
                   IF #LT_Crane_Feed THEN
                       #Loading_to_Crane_Conveyor := FALSE;
                       #StackerCrane_1_Left := TRUE;
                       #State := 1;
                   END_IF;
               END_IF;
               // 1 - Pick up pallet
           1:
               IF #StackerCrane_1_Left_Limit THEN
                   // Lift pallet
                   #StackerCrane_1_Lift := TRUE;
                   // Retract forks
                   #StackerCrane_1_Left := FALSE;
                   #State := 2;
               END_IF;
               // 2 - Wait until forks reach MIDDLE
           2:
               IF #StackerCrane_1_Middle_Limit THEN
                   #StackerCrane_1_Target_1_Position := #NextPosition;
                   #MovementStarted := FALSE;
                   #State := 3;
               END_IF;
               // 3 - Move X/Z and extend forks RIGHT
           3:
               #StackerCrane_1_Target_1_Position := #NextPosition;
               IF #StackerCrane_1_Moving_X
                   OR #StackerCrane_1_Moving_Z THEN
                   #MovementStarted := TRUE;
               END_IF;
               IF #MovementStarted
                   AND NOT #StackerCrane_1_Moving_X
                   AND NOT #StackerCrane_1_Moving_Z THEN
                   #MovementStarted := FALSE;
                   // Extend forks into rack
                   #StackerCrane_1_Right := TRUE;
               END_IF;
               IF #StackerCrane_1_Right_Limit THEN
                   // Lower pallet onto rack
                   // Lift remains FALSE from this point
                   #StackerCrane_1_Lift := FALSE;
                   #State := 4;
               END_IF;
               // 4 - Wait for pallet to settle
           4:
               #StackerCrane_1_Target_1_Position := #NextPosition;
               IF #TimerDeposit.Q THEN
                   // Retract forks only after pallet has settled
                   #StackerCrane_1_Right := FALSE;
                   #State := 5;
               END_IF;
               // 5 - Wait until forks reach MIDDLE
           5:
               #StackerCrane_1_Target_1_Position := #NextPosition;
               IF #StackerCrane_1_Middle_Limit THEN
                   #StackerCrane_1_Target_1_Position := 55;
                   #MovementStarted := FALSE;
                   #State := 6;
               END_IF;
               // 6 - Return to REST
           6:
               #StackerCrane_1_Target_1_Position := 55;
               IF #StackerCrane_1_Moving_X
                   OR #StackerCrane_1_Moving_Z THEN
                   #MovementStarted := TRUE;
               END_IF;
               IF #MovementStarted
                   AND NOT #StackerCrane_1_Moving_X
                   AND NOT #StackerCrane_1_Moving_Z THEN
                   #StackerCrane_1_Target_1_Position := 0;
                   #MovementStarted := FALSE;
                   IF #NextPosition < 54 THEN
                       #NextPosition := #NextPosition + 1;
                       #State := 0;
                   ELSE
                       #State := 7;
                   END_IF;
               END_IF;
               // 7 - Warehouse full
           7:
               #StackerCrane_1_Target_1_Position := 0;
           ELSE
               #State := 0;
       END_CASE;
   END_IF;
END_FUNCTION_BLOCK

// folder: 07_HMI

FUNCTION "FC_HMI_Status" : Bool   // FC3, SCL
{ S7_Optimized_Access := 'TRUE' }
VERSION : 0.1
BEGIN
   // 0 = Idle 1 = Ready 2 = Busy
   // Lid status
   IF "FB_LidCenter_DB".Busy THEN
       "DB_Global".HMI_LidStatus := 2;
   ELSIF "FB_LidCenter_DB".Ready THEN
       "DB_Global".HMI_LidStatus := 1;
   ELSE
       "DB_Global".HMI_LidStatus := 0;
   END_IF;

   // Base status
   IF "FB_BaseCenter_DB".Busy THEN
       "DB_Global".HMI_BaseStatus := 2;
   ELSIF "FB_BaseCenter_DB".Ready THEN
       "DB_Global".HMI_BaseStatus := 1;
   ELSE
       "DB_Global".HMI_BaseStatus := 0;
   END_IF;

   // Warehouse status
   IF "FB_Warehouse_DB".WarehouseFull THEN
       "DB_Global".HMI_WarehouseStatus := 3;
   ELSIF "FB_Warehouse_DB".Busy THEN
       "DB_Global".HMI_WarehouseStatus := 2;
   ELSIF "FB_Warehouse_DB".Ready THEN
       "DB_Global".HMI_WarehouseStatus := 1;
   ELSE
       "DB_Global".HMI_WarehouseStatus := 0;
   END_IF;

   // Warehouse full status
   "DB_Global".Warehouse_Full := "FB_Warehouse_DB".WarehouseFull;

   // Warehouse full alarm
   "DB_Global".HMI_AlarmWord.%X0 := "FB_Warehouse_DB".WarehouseFull;

   // Warehouse alarm acknowledgement
   IF "DB_Global".HMI_AckWord.%X0 THEN
       "FACTORY I/O (Reset)" := TRUE;
       "DB_Global".HMI_AckWord.%X0 := FALSE;
   END_IF;

   // Total packages stored in Warehouse
   "DB_Global".HMI_TotalPackages := "DB_Global".HMI_OccupiedPositions * 4;

   // FC executed successfully
   #FC_HMI_Status := TRUE;
END_FUNCTION

(* ===== HMI "HMI_RT_1" =====
system functions are stored by id; their names below are inferred from use
connection "HMI_Verbindung_1": ETHERNET, SMART_S7_1500_OMS

HMI tags "Standard-Variablentabelle"
   "Variable_Bildnummer" : UInt, internal
   "Plant_Enabled_HMI" : Bool = PLC DB_Global.Plant_Enabled AT %DB1.DBX0.0, 1 s
   "Reset_HMI" : Bool = PLC "FACTORY I/O (Reset)" AT %I4.2, 1 s
   "Production_Lid_Status_HMI" : USInt = PLC DB_Global.HMI_LidStatus AT %DB1.DBX0.0, 1 s
   "Production_Base_Status_HMI" : USInt = PLC DB_Global.HMI_BaseStatus AT %DB1.DBB0, 1 s
   "Warehouse_Status_HMI" : USInt = PLC DB_Global.HMI_WarehouseStatus AT %DB1.DBB0, 1 s
   "HMI_OccupiedPositions" : DInt = PLC DB_Global.HMI_OccupiedPositions AT %DB1.DBB0, 1 s
   "HMI_FreePositions" : DInt = PLC DB_Global.HMI_FreePositions AT %DB1.DBB0, 1 s
   "HMI_TotalPackages" : DInt = PLC DB_Global.HMI_TotalPackages AT %DB1.DBW0, 1 s
   "HMI_WarehouseFull" : Bool = PLC DB_Global.Warehouse_Full AT %DB1.DBD0, 1 s
   "HMI_AlarmWord" : Word = PLC DB_Global.HMI_AlarmWord AT %DB1.DBW0, 1 s
   "HMI_AckWord" : Word = PLC DB_Global.HMI_AckWord AT %DB1.DBW0, 1 s
   "HMI_Count_BlueBlue" : DInt = PLC FB_ProductTracking_DB.Count_BlueBlue AT %DB1.DBD0, 1 s
   "HMI_Count_BlueGreen" : DInt = PLC FB_ProductTracking_DB.Count_BlueGreen AT %DB1.DBD0, 1 s
   "HMI_Count_BlueMetal" : DInt = PLC FB_ProductTracking_DB.Count_BlueMetal AT %DB1.DBD0, 1 s
   "HMI_Count_GreenGreen" : DInt = PLC FB_ProductTracking_DB.Count_GreenGreen AT %DB1.DBD0, 1 s
   "HMI_Count_GreenMetal" : DInt = PLC FB_ProductTracking_DB.Count_GreenMetal AT %DB1.DBD0, 1 s
   "HMI_Count_MetalBlue" : DInt = PLC FB_ProductTracking_DB.Count_MetalBlue AT %DB1.DBD0, 1 s
   "HMI_Count_MetalGreen" : DInt = PLC FB_ProductTracking_DB.Count_MetalGreen AT %DB1.DBD0, 1 s
   "HMI_Count_MetalMetal" : DInt = PLC FB_ProductTracking_DB.Count_MetalMetal AT %DB1.DBD0, 1 s
   "HMI_Count_GreenBlue" : DInt = PLC FB_ProductTracking_DB.Count_GreenBlue AT %DB1.DBD0, 1 s

discrete alarms
   1: 'Warehouse storage full! System will restart and Warehouse will be unloaded after message acknowledgement!', class Errors, trigger "HMI_AlarmWord" bit 0

Template "Vorlage_1" 800x480
   Button "Exit" at 722,440 size 55x39; TextOff 'Exit'; PictureOff "ExitRuntime_KTP900_Basic_PN_TR"; PictureOn "ExitRuntime_KTP900_Basic_PN_TR"
      on Release: StopRuntime(0)
   Button "Log on" at 622,440 size 55x39; TextOff 'Log on'; PictureOff "Login_KTP900_Basic_PN_TR"; PictureOn "Login_KTP900_Basic_PN_TR"
      on Release: function_a2a04561()
   Button "Language" at 522,440 size 55x39; TextOff 'Language'; PictureOff "ToggleLanguage_KTP900_Basic_PN_TR"; PictureOn "ToggleLanguage_KTP900_Basic_PN_TR"
      on Release: function_fb9197e8(-1)
   Button "Template_Button" at 422,440 size 55x39; TextOff 'Text'
   Button "Template_Button_1" at 322,440 size 55x39; TextOff 'Text'
   Button "Template_Button_2" at 222,440 size 55x39; TextOff 'Text'
   Button "Start screen" at 122,440 size 55x39; TextOff 'Start screen'; PictureOff "NavigateHome_KTP900_Basic_PN_TR"; PictureOn "NavigateHome_KTP900_Basic_PN_TR"
      on Release: ActivateScreen("Grundbild", 0)
   Button "Alarms" at 22,440 size 55x39; TextOff 'Alarms'; PictureOff "AlarmDisplay_KTP900_Basic_PN_TR"; PictureOn "AlarmDisplay_KTP900_Basic_PN_TR"
      on Release: function_ef3f5d25("Meldefenster_Nichtquittiert", -1)
   SymbolicIOField "Symbolisches_EA_Feld_Bild" at 73,7 size 620x26; TextOff '0'; TextOn '1'; TextList "TextList_ScreenNames"
      ProcessValue <- "Variable_Bildnummer"
      on Change: ActivateScreenByNumber("Variable_Bildnummer", 0)
   DateTimeField "HmiScreenItemData" at 695,20 size 105x20
   DateTimeField "HmiScreenItemData_1" at 695,0 size 105x20
   GraphicView "Logo" at 0,0 size 71x40; Picture "Logo of HMI_1"

screen "Grundbild" 800x480, template "Vorlage_1"
   on GenerateScreen: SetTag("Variable_Bildnummer", 1)
   TextField "HmiScreenItemData_4" at 80,226 size 640x22; Text 'Welcome to HMI_1 (KTP900 Basic+ PN)!'
   Button "HmiScreenItemData" at 36,76 size 159x47; TextOff 'Plant Control'; PictureOff "Navigates to menu1 for KTP900 Basic+ PN 17.0.0.0"; PictureOn "Navigates to menu1 for KTP900 Basic+ PN 17.0.0.0"
      on Release: ActivateScreen("Plant Control", 0)
   Button "HmiScreenItemData_5" at 36,136 size 159x47; TextOff 'System screens'; PictureOff "Navigates to Systembilder for KTP900 Basic+ PN 17.0.0.0"; PictureOn "Navigates to Systembilder for KTP900 Basic+ PN 17.0.0.0"
      on Release: ActivateScreen("Systembilder", 0)

screen "Plant Control" 800x480, template "Vorlage_1"
   on GenerateScreen: SetTag("Variable_Bildnummer", 2)
   Button "Back" at 1,41 size 159x47; TextOff 'Back'
      on Release: ActivateScreen("Grundbild", 0)
   Button "Schaltfläche_1" at 173,97 size 96x32; TextOff 'Start'
      on Press: SetBit("Plant_Enabled_HMI")
      Appearance <- "Plant_Enabled_HMI"
   Button "Schaltfläche_2" at 279,97 size 96x32; TextOff 'Stop'
      on Press: ResetBit("Plant_Enabled_HMI")
      Appearance <- "Plant_Enabled_HMI"
   Button "Schaltfläche_3" at 382,96 size 96x32; TextOff 'Reset'
      on Press: SetBit("Reset_HMI")
      Appearance <- "Reset_HMI"
   TextField "Textfeld_3" at 41,94 size 85x20; Text 'PRODUCTION'
   TextField "Textfeld_2" at 37,118 size 23x20; Text 'Lid'
   TextField "Textfeld_4" at 28,141 size 36x20; Text 'Base'
   IOField "EA-Feld_1" at 63,327 size 32x32; FormatPattern 99
      ProcessValue <- "HMI_TotalPackages"
   TextField "Textfeld_7" at 19,305 size 116x20; Text 'TOTAL PACKAGES'
   TextField "Textfeld_8" at 14,189 size 159x20; Text 'WAREHOUSE STORAGE'
   TextField "Textfeld_9" at 19,217 size 68x20; Text 'Occupied:'
   IOField "EA-Feld_2" at 93,210 size 31x32; FormatPattern 99
      ProcessValue <- "HMI_OccupiedPositions"
   TextField "Textfeld_10" at 20,261 size 38x20; Text 'Free:'
   IOField "EA-Feld_3" at 94,254 size 32x32; FormatPattern 99
      ProcessValue <- "HMI_FreePositions"
   Button "Schaltfläche_6" at 426,349 size 27x32; TextOff '1'
      Appearance <- "HMI_OccupiedPositions"
   Button "Schaltfläche_7" at 401,349 size 27x32; TextOff '2'
      Appearance <- "HMI_OccupiedPositions"
   Button "Schaltfläche_8" at 376,349 size 27x32; TextOff '3'
      Appearance <- "HMI_OccupiedPositions"
   Button "Schaltfläche_9" at 352,349 size 27x32; TextOff '4'
      Appearance <- "HMI_OccupiedPositions"
   Button "Schaltfläche_10" at 327,349 size 27x32; TextOff '5'
      Appearance <- "HMI_OccupiedPositions"
   Button "Schaltfläche_11" at 302,349 size 27x32; TextOff '6'
      Appearance <- "HMI_OccupiedPositions"
   Button "Schaltfläche_12" at 278,349 size 27x32; TextOff '7'
      Appearance <- "HMI_OccupiedPositions"
   Button "Schaltfläche_13" at 253,349 size 27x32; TextOff '8'
      Appearance <- "HMI_OccupiedPositions"
   Button "Schaltfläche_14" at 228,349 size 27x32; TextOff '9'
      Appearance <- "HMI_OccupiedPositions"
   Button "Schaltfläche_15" at 426,319 size 27x32; TextOff '10'
      Appearance <- "HMI_OccupiedPositions"
   Button "Schaltfläche_16" at 402,319 size 27x32; TextOff '11'
      Appearance <- "HMI_OccupiedPositions"
   Button "Schaltfläche_17" at 377,319 size 27x32; TextOff '12'
      Appearance <- "HMI_OccupiedPositions"
   Button "Schaltfläche_18" at 352,319 size 27x32; TextOff '13'
      Appearance <- "HMI_OccupiedPositions"
   Button "Schaltfläche_19" at 327,319 size 27x32; TextOff '14'
      Appearance <- "HMI_OccupiedPositions"
   Button "Schaltfläche_20" at 303,319 size 27x32; TextOff '15'
      Appearance <- "HMI_OccupiedPositions"
   Button "Schaltfläche_21" at 278,319 size 27x32; TextOff '16'
      Appearance <- "HMI_OccupiedPositions"
   Button "Schaltfläche_22" at 253,319 size 27x32; TextOff '17'
      Appearance <- "HMI_OccupiedPositions"
   Button "Schaltfläche_23" at 228,319 size 27x32; TextOff '18'
      Appearance <- "HMI_OccupiedPositions"
   Circle "Kreis_2" at 70,118 size 16x16
      Appearance <- "Production_Lid_Status_HMI"
   Circle "Kreis_4" at 70,141 size 16x16
      Appearance <- "Production_Base_Status_HMI"
   Button "Schaltfläche_4" at 426,289 size 27x32; TextOff '19'
      Appearance <- "HMI_OccupiedPositions"
   Button "Schaltfläche_5" at 401,289 size 27x32; TextOff '20'
      Appearance <- "HMI_OccupiedPositions"
   Button "Schaltfläche_24" at 376,289 size 27x32; TextOff '21'
      Appearance <- "HMI_OccupiedPositions"
   Button "Schaltfläche_25" at 352,289 size 26x32; TextOff '22'
      Appearance <- "HMI_OccupiedPositions"
   Button "Schaltfläche_26" at 327,289 size 27x32; TextOff '23'
      Appearance <- "HMI_OccupiedPositions"
   Button "Schaltfläche_27" at 302,289 size 27x32; TextOff '24'
      Appearance <- "HMI_OccupiedPositions"
   Button "Schaltfläche_28" at 278,289 size 27x32; TextOff '25'
      Appearance <- "HMI_OccupiedPositions"
   Button "Schaltfläche_29" at 253,289 size 27x32; TextOff '26'
      Appearance <- "HMI_OccupiedPositions"
   Button "Schaltfläche_30" at 228,289 size 27x32; TextOff '27'
      Appearance <- "HMI_OccupiedPositions"
   Button "Schaltfläche_31" at 426,261 size 27x32; TextOff '28'
      Appearance <- "HMI_OccupiedPositions"
   Button "Schaltfläche_32" at 401,261 size 27x32; TextOff '29'
      Appearance <- "HMI_OccupiedPositions"
   Button "Schaltfläche_33" at 376,261 size 27x32; TextOff '30'
      Appearance <- "HMI_OccupiedPositions"
   Button "Schaltfläche_34" at 352,261 size 27x32; TextOff '31'
      Appearance <- "HMI_OccupiedPositions"
   Button "Schaltfläche_35" at 327,261 size 27x32; TextOff '32'
      Appearance <- "HMI_OccupiedPositions"
   Button "Schaltfläche_36" at 302,261 size 27x32; TextOff '33'
      Appearance <- "HMI_OccupiedPositions"
   Button "Schaltfläche_37" at 277,261 size 27x32; TextOff '34'
      Appearance <- "HMI_OccupiedPositions"
   Button "Schaltfläche_38" at 253,261 size 27x32; TextOff '35'
      Appearance <- "HMI_OccupiedPositions"
   Button "Schaltfläche_39" at 228,261 size 27x32; TextOff '36'
      Appearance <- "HMI_OccupiedPositions"
   Button "Schaltfläche_40" at 426,231 size 27x32; TextOff '37'
      Appearance <- "HMI_OccupiedPositions"
   Button "Schaltfläche_41" at 401,231 size 27x32; TextOff '38'
      Appearance <- "HMI_OccupiedPositions"
   Button "Schaltfläche_42" at 377,231 size 27x32; TextOff '39'
      Appearance <- "HMI_OccupiedPositions"
   Button "Schaltfläche_43" at 352,231 size 27x32; TextOff '40'
      Appearance <- "HMI_OccupiedPositions"
   Button "Schaltfläche_44" at 327,231 size 27x32; TextOff '41'
      Appearance <- "HMI_OccupiedPositions"
   Button "Schaltfläche_45" at 302,231 size 27x32; TextOff '42'
      Appearance <- "HMI_OccupiedPositions"
   Button "Schaltfläche_46" at 278,231 size 27x32; TextOff '43'
      Appearance <- "HMI_OccupiedPositions"
   Button "Schaltfläche_47" at 253,231 size 27x32; TextOff '44'
      Appearance <- "HMI_OccupiedPositions"
   Button "Schaltfläche_48" at 228,231 size 27x32; TextOff '45'
      Appearance <- "HMI_OccupiedPositions"
   Button "Schaltfläche_49" at 426,201 size 27x32; TextOff '46'
      Appearance <- "HMI_OccupiedPositions"
   Button "Schaltfläche_50" at 401,201 size 27x32; TextOff '47'
      Appearance <- "HMI_OccupiedPositions"
   Button "Schaltfläche_51" at 376,201 size 27x32; TextOff '48'
      Appearance <- "HMI_OccupiedPositions"
   Button "Schaltfläche_52" at 352,201 size 27x32; TextOff '49'
      Appearance <- "HMI_OccupiedPositions"
   Button "Schaltfläche_53" at 327,201 size 27x32; TextOff '50'
      Appearance <- "HMI_OccupiedPositions"
   Button "Schaltfläche_54" at 302,201 size 27x32; TextOff '51'
      Appearance <- "HMI_OccupiedPositions"
   Button "Schaltfläche_55" at 278,201 size 27x32; TextOff '52'
      Appearance <- "HMI_OccupiedPositions"
   Button "Schaltfläche_56" at 253,201 size 27x32; TextOff '53'
      Appearance <- "HMI_OccupiedPositions"
   Button "Schaltfläche_57" at 228,201 size 27x32; TextOff '54'
      Appearance <- "HMI_OccupiedPositions"
   TextField "Textfeld_1" at 277,179 size 115x20; Text 'Warehouse Slots'
   AlarmView "Meldeanzeige_1" at 173,35 size 600x59
      Visibility <- "HMI_AlarmWord"
   TextField "Textfeld_5" at 595,204 size 56x20; Text 'Blue'
   TextField "Textfeld_6" at 544,236 size 56x20; Text 'Blue'
   TextField "Textfeld_11" at 642,202 size 43x20; Text 'Green'
   TextField "Textfeld_12" at 690,202 size 41x20; Text 'Metal'
   TextField "Textfeld_13" at 544,274 size 43x20; Text 'Green'
   TextField "Textfeld_14" at 544,308 size 61x20; Text 'Metal'
   IOField "EA-Feld_4" at 595,232 size 40x32; FormatPattern 999
      ProcessValue <- "HMI_Count_BlueBlue"
   IOField "EA-Feld_5" at 690,231 size 40x32; FormatPattern 999
      ProcessValue <- "HMI_Count_BlueMetal"
   IOField "EA-Feld_6" at 642,232 size 40x32; FormatPattern 999
      ProcessValue <- "HMI_Count_BlueGreen"
   IOField "EA-Feld_7" at 595,269 size 40x32; FormatPattern 999
      ProcessValue <- "HMI_Count_GreenBlue"
   IOField "EA-Feld_8" at 690,268 size 40x32; FormatPattern 999
      ProcessValue <- "HMI_Count_GreenMetal"
   IOField "EA-Feld_9" at 642,269 size 40x32; FormatPattern 999
      ProcessValue <- "HMI_Count_GreenGreen"
   IOField "EA-Feld_10" at 595,306 size 40x32; FormatPattern 999
      ProcessValue <- "HMI_Count_MetalBlue"
   IOField "EA-Feld_11" at 690,305 size 40x32; FormatPattern 999
      ProcessValue <- "HMI_Count_MetalMetal"
   IOField "EA-Feld_12" at 642,306 size 40x32; FormatPattern 999
      ProcessValue <- "HMI_Count_MetalGreen"
   TextField "Textfeld_15" at 622,183 size 68x20; Text 'Lid Colour'
   TextField "Textfeld_16" at 500,273 size 36x20; Text 'Base'
   TextField "Textfeld_17" at 493,289 size 46x20; Text 'Colour'

screen "Systembilder" 800x480, template "Vorlage_1"
   on GenerateScreen: SetTag("Variable_Bildnummer", 6)
   Button "Back" at 1,41 size 159x47; TextOff 'Back'
      on Release: ActivateScreen("Grundbild", 0)
   Button "HmiScreenItemData" at 36,135 size 159x47; TextOff 'SIMATIC PLC system diagnos...'; PictureOff "Navigates to SIMATIC PLC Systemdiagnose for KTP900 Basic+ PN 17.0.0.0"; PictureOn "Navigates to SIMATIC PLC Systemdiagnose for KTP900 Basic+ PN 17.0.0.0"
      on Release: ActivateScreen("SIMATIC PLC Systemdiagnose", 0)
   Button "HmiScreenItemData_1" at 36,194 size 159x47; TextOff 'Project information'; PictureOff "Navigates to Projektinformationen for KTP900 Basic+ PN 17.0.0.0"; PictureOn "Navigates to Projektinformationen for KTP900 Basic+ PN 17.0.0.0"
      on Release: ActivateScreen("Projektinformationen", 0)
   Button "HmiScreenItemData_2" at 36,253 size 159x47; TextOff 'User administration'; PictureOff "Navigates to Benutzerverwaltung for KTP900 Basic+ PN 17.0.0.0"; PictureOn "Navigates to Benutzerverwaltung for KTP900 Basic+ PN 17.0.0.0"
      on Release: ActivateScreen("Benutzerverwaltung", 0)
   Button "HmiScreenItemData_3" at 36,312 size 159x47; TextOff 'System information'; PictureOff "Navigates to Systeminformationen for KTP900 Basic+ PN 17.0.0.0"; PictureOn "Navigates to Systeminformationen for KTP900 Basic+ PN 17.0.0.0"
      on Release: ActivateScreen("Systeminformationen", 0)
   Button "HmiScreenItemData_4" at 36,371 size 159x47; TextOff 'Different jobs'; PictureOff "Navigates to Verschiedene Aufgaben for KTP900 Basic+ PN 17.0.0.0"; PictureOn "Navigates to Verschiedene Aufgaben for KTP900 Basic+ PN 17.0.0.0"
      on Release: ActivateScreen("Verschiedene Aufgaben", 0)

screen "SIMATIC PLC Systemdiagnose" 800x480, template "Vorlage_1"
   on GenerateScreen: SetTag("Variable_Bildnummer", 7)
   SysDiagControl "HmiScreenItemData" at 1,89 size 796x343
   Button "Back" at 1,41 size 159x47; TextOff 'Back'
      on Release: ActivateScreen("Systembilder", 0)

screen "Projektinformationen" 800x480, template "Vorlage_1"
   on GenerateScreen: SetTag("Variable_Bildnummer", 8)
   TextField "HmiScreenItemData" at 35,91 size 171x28; Text 'Project name:'
   TextField "HmiScreenItemData_1" at 241,91 size 524x28; Text 'Abschulss_Projekt'
   TextField "HmiScreenItemData_2" at 35,121 size 171x28; Text 'Created on:'
   TextField "HmiScreenItemData_3" at 241,121 size 524x28; Text '07.04.2016 11:51:36'
   TextField "HmiScreenItemData_4" at 35,151 size 171x28; Text 'Author:'
   TextField "HmiScreenItemData_5" at 241,151 size 524x28; Text 'Matthias Habermann'
   TextField "HmiScreenItemData_6" at 35,181 size 171x28; Text 'Description:'
   TextField "HmiScreenItemData_7" at 241,181 size 524x28; Text '(not configured)'
   Button "Back" at 1,41 size 159x47; TextOff 'Back'
      on Release: ActivateScreen("Systembilder", 0)

screen "Benutzerverwaltung" 800x480, template "Vorlage_1"
   on GenerateScreen: SetTag("Variable_Bildnummer", 9)
   UserView "HmiScreenItemData" at 1,89 size 796x343
   Button "Back" at 1,41 size 159x47; TextOff 'Back'
      on Release: ActivateScreen("Systembilder", 0)

screen "Systeminformationen" 800x480, template "Vorlage_1"
   on GenerateScreen: SetTag("Variable_Bildnummer", 10)
   TextField "HmiScreenItemData" at 35,91 size 171x28; Text 'HMI device type:'
   TextField "HmiScreenItemData_1" at 241,91 size 524x28; Text 'KTP900 Basic+ PN 17.0.0.0'
   TextField "HmiScreenItemData_2" at 35,121 size 171x28; Text 'Connection:'
   TextField "HmiScreenItemData_3" at 241,121 size 524x28; Text 'PROFINET (X1)'
   TextField "HmiScreenItemData_4" at 35,151 size 171x28; Text 'PLC:'
   TextField "HmiScreenItemData_5" at 241,151 size 524x28; Text 'SIMATIC S7 1500'
   Button "Back" at 1,41 size 159x47; TextOff 'Back'
      on Release: ActivateScreen("Systembilder", 0)

screen "Verschiedene Aufgaben" 800x480, template "Vorlage_1"
   on GenerateScreen: SetTag("Variable_Bildnummer", 11)
   Button "Online" at 36,135 size 159x47; TextOff 'Online'
      on Release: function_bb44b551(0)
   Button "Offline" at 36,194 size 159x47; TextOff 'Offline'
      on Release: function_bb44b551(1)
   Button "Transfer" at 36,253 size 159x47; TextOff 'Transfer'
      on Release: function_bb44b551(2)
   Button "Toggle language" at 36,312 size 159x47; TextOff 'Toggle language'
      on Release: function_fb9197e8(-1)
   Button "Stop Runtime" at 36,371 size 159x47; TextOff 'Stop Runtime'
      on Release: StopRuntime(0)
   Button "Back" at 1,41 size 159x47; TextOff 'Back'
      on Release: ActivateScreen("Systembilder", 0)
*)